(*	=====	LUC	[1]	==========	=	=	*)
		If NOT emC_PPC[PPCNum].LuC[1].In.ComFault	THEN
			emC_PPC[PPCNum].Summary.GCFaultSt	:=	emC_PPC[PPCNum].Summary.GCFaultSt	OR	emC_PPC[PPCNum].LuC[1].In.GCFaultSt	;
			emC_PPC[PPCNum].Summary.NonCriticalAlarm	:=	emC_PPC[PPCNum].Summary.NonCriticalAlarm	OR	emC_PPC[PPCNum].LuC[1].In.NonCriticalAlarm	;
			emC_PPC[PPCNum].Summary.CriticalAlarm	:=	emC_PPC[PPCNum].Summary.CriticalAlarm	OR	emC_PPC[PPCNum].LuC[1].In.CriticalAlarm	;
			emC_PPC[PPCNum].Summary.Warning	:=	emC_PPC[PPCNum].Summary.Warning	OR	emC_PPC[PPCNum].LuC[1].In.Warning	;
			emC_PPC[PPCNum].Summary.StoppingSt	:=	emC_PPC[PPCNum].Summary.StoppingSt	OR	emC_PPC[PPCNum].LuC[1].In.StoppingSt	;
			emC_PPC[PPCNum].Summary.BlackSys	:=	emC_PPC[PPCNum].Summary.BlackSys	OR	emC_PPC[PPCNum].LuC[1].In.BlackSys	;
		END_IF;
		If NOT emC_PPC[PPCNum].LuC[1].In.ComFault	THEN
			emC_PPC[PPCNum].Summary.ComFaultCnt	:=	emC_PPC[PPCNum].Summary.ComFaultCnt	+	1	;
		END_IF;
		If NOT emC_PPC[PPCNum].LuC[1].In.ComFault AND	emC_PPC[PPCNum].LuC[1].In.OnlineSt 	THEN
		
				emC_PPC[PPCNum].Summary.OnlineCnt	:=	emC_PPC[PPCNum].Summary.OnlineCnt	+	1	;
								
				emC_PPC[PPCNum].Summary.AvgTempAct	:=	(emC_PPC[PPCNum].Summary.AvgTempAct	+	emC_PPC[PPCNum].LuC[1].In.TempAct)/INT_TO_REAL(emC_PPC[PPCNum].Summary.OnlineCnt)	;
				emC_PPC[PPCNum].Summary.TotBatPNomMaxAct	:=	emC_PPC[PPCNum].Summary.TotBatPNomMaxAct	+	emC_PPC[PPCNum].LuC[1].In.BatPNomMaxAct	;
				emC_PPC[PPCNum].Summary.TotBatPNomMinAct	:=	emC_PPC[PPCNum].Summary.TotBatPNomMinAct	+	emC_PPC[PPCNum].LuC[1].In.BatPNomMinAct	;
				emC_PPC[PPCNum].Summary.AvgSocPct	:=	(emC_PPC[PPCNum].Summary.AvgSocPct	+	emC_PPC[PPCNum].LuC[1].In.SocPctAct)/INT_TO_REAL(emC_PPC[PPCNum].Summary.OnlineCnt)	;
				emC_PPC[PPCNum].Summary.AvgUAct	:=	(emC_PPC[PPCNum].Summary.AvgUAct	+	emC_PPC[PPCNum].LuC[1].In.UAct)/INT_TO_REAL(emC_PPC[PPCNum].Summary.OnlineCnt)	;
				emC_PPC[PPCNum].Summary.AvgFAct	:=	(emC_PPC[PPCNum].Summary.AvgFAct	+	emC_PPC[PPCNum].LuC[1].In.FAct)/INT_TO_REAL(emC_PPC[PPCNum].Summary.OnlineCnt)	;
				emC_PPC[PPCNum].Summary.TotPAct	:=	emC_PPC[PPCNum].Summary.TotPAct	+	emC_PPC[PPCNum].LuC[1].In.PAct	;
				emC_PPC[PPCNum].Summary.TotQAct	:=	emC_PPC[PPCNum].Summary.TotQAct	+	emC_PPC[PPCNum].LuC[1].In.QAct	;
		
		END_IF	;	
								
								
(*	=====	LUC	[2]	==========	=	=	*)
		If NOT emC_PPC[PPCNum].LuC[2].In.ComFault	THEN						
			emC_PPC[PPCNum].Summary.GCFaultSt	:=	emC_PPC[PPCNum].Summary.GCFaultSt	OR	emC_PPC[PPCNum].LuC[2].In.GCFaultSt	;	
			emC_PPC[PPCNum].Summary.NonCriticalAlarm	:=	emC_PPC[PPCNum].Summary.NonCriticalAlarm	OR	emC_PPC[PPCNum].LuC[2].In.NonCriticalAlarm	;	
			emC_PPC[PPCNum].Summary.CriticalAlarm	:=	emC_PPC[PPCNum].Summary.CriticalAlarm	OR	emC_PPC[PPCNum].LuC[2].In.CriticalAlarm	;	
			emC_PPC[PPCNum].Summary.Warning	:=	emC_PPC[PPCNum].Summary.Warning	OR	emC_PPC[PPCNum].LuC[2].In.Warning	;	
			emC_PPC[PPCNum].Summary.StoppingSt	:=	emC_PPC[PPCNum].Summary.StoppingSt	OR	emC_PPC[PPCNum].LuC[2].In.StoppingSt	;	
			emC_PPC[PPCNum].Summary.BlackSys	:=	emC_PPC[PPCNum].Summary.BlackSys	OR	emC_PPC[PPCNum].LuC[2].In.BlackSys	;	
		END_IF;							
		If NOT emC_PPC[PPCNum].LuC[2].In.ComFault	THEN						
			emC_PPC[PPCNum].Summary.ComFaultCnt	:=	emC_PPC[PPCNum].Summary.ComFaultCnt	+	1	;	
		END_IF;							
		If NOT emC_PPC[PPCNum].LuC[2].In.ComFault AND	emC_PPC[PPCNum].LuC[2].In.OnlineSt 	THEN					
							
				emC_PPC[PPCNum].Summary.OnlineCnt	:=	emC_PPC[PPCNum].Summary.OnlineCnt	+	1	;
							
				emC_PPC[PPCNum].Summary.AvgTempAct	:=	(emC_PPC[PPCNum].Summary.AvgTempAct	+	emC_PPC[PPCNum].LuC[2].In.TempAct)/INT_TO_REAL(emC_PPC[PPCNum].Summary.OnlineCnt)	;
				emC_PPC[PPCNum].Summary.TotBatPNomMaxAct	:=	emC_PPC[PPCNum].Summary.TotBatPNomMaxAct	+	emC_PPC[PPCNum].LuC[2].In.BatPNomMaxAct	;
				emC_PPC[PPCNum].Summary.TotBatPNomMinAct	:=	emC_PPC[PPCNum].Summary.TotBatPNomMinAct	+	emC_PPC[PPCNum].LuC[2].In.BatPNomMinAct	;
				emC_PPC[PPCNum].Summary.AvgSocPct	:=	(emC_PPC[PPCNum].Summary.AvgSocPct	+	emC_PPC[PPCNum].LuC[2].In.SocPctAct)/INT_TO_REAL(emC_PPC[PPCNum].Summary.OnlineCnt)	;
				emC_PPC[PPCNum].Summary.AvgUAct	:=	(emC_PPC[PPCNum].Summary.AvgUAct	+	emC_PPC[PPCNum].LuC[2].In.UAct)/INT_TO_REAL(emC_PPC[PPCNum].Summary.OnlineCnt)	;
				emC_PPC[PPCNum].Summary.AvgFAct	:=	(emC_PPC[PPCNum].Summary.AvgFAct	+	emC_PPC[PPCNum].LuC[2].In.FAct)/INT_TO_REAL(emC_PPC[PPCNum].Summary.OnlineCnt)	;
				emC_PPC[PPCNum].Summary.TotPAct	:=	emC_PPC[PPCNum].Summary.TotPAct	+	emC_PPC[PPCNum].LuC[2].In.PAct	;
				emC_PPC[PPCNum].Summary.TotQAct	:=	emC_PPC[PPCNum].Summary.TotQAct	+	emC_PPC[PPCNum].LuC[2].In.QAct	;
							
		END_IF	;	
								
					
(*	=====	LUC	[3]	==========	=	=	*)
		If NOT emC_PPC[PPCNum].LuC[3].In.ComFault	THEN						
			emC_PPC[PPCNum].Summary.GCFaultSt	:=	emC_PPC[PPCNum].Summary.GCFaultSt	OR	emC_PPC[PPCNum].LuC[3].In.GCFaultSt	;	
			emC_PPC[PPCNum].Summary.NonCriticalAlarm	:=	emC_PPC[PPCNum].Summary.NonCriticalAlarm	OR	emC_PPC[PPCNum].LuC[3].In.NonCriticalAlarm	;	
			emC_PPC[PPCNum].Summary.CriticalAlarm	:=	emC_PPC[PPCNum].Summary.CriticalAlarm	OR	emC_PPC[PPCNum].LuC[3].In.CriticalAlarm	;	
			emC_PPC[PPCNum].Summary.Warning	:=	emC_PPC[PPCNum].Summary.Warning	OR	emC_PPC[PPCNum].LuC[3].In.Warning	;	
			emC_PPC[PPCNum].Summary.StoppingSt	:=	emC_PPC[PPCNum].Summary.StoppingSt	OR	emC_PPC[PPCNum].LuC[3].In.StoppingSt	;	
			emC_PPC[PPCNum].Summary.BlackSys	:=	emC_PPC[PPCNum].Summary.BlackSys	OR	emC_PPC[PPCNum].LuC[3].In.BlackSys	;	
		END_IF;							
		If NOT emC_PPC[PPCNum].LuC[3].In.ComFault	THEN						
			emC_PPC[PPCNum].Summary.ComFaultCnt	:=	emC_PPC[PPCNum].Summary.ComFaultCnt	+	1	;	
		END_IF;							
		If NOT emC_PPC[PPCNum].LuC[3].In.ComFault AND	emC_PPC[PPCNum].LuC[3].In.OnlineSt 	THEN					
							
				emC_PPC[PPCNum].Summary.OnlineCnt	:=	emC_PPC[PPCNum].Summary.OnlineCnt	+	1	;
							
				emC_PPC[PPCNum].Summary.AvgTempAct	:=	(emC_PPC[PPCNum].Summary.AvgTempAct	+	emC_PPC[PPCNum].LuC[3].In.TempAct)/INT_TO_REAL(emC_PPC[PPCNum].Summary.OnlineCnt)	;
				emC_PPC[PPCNum].Summary.TotBatPNomMaxAct	:=	emC_PPC[PPCNum].Summary.TotBatPNomMaxAct	+	emC_PPC[PPCNum].LuC[3].In.BatPNomMaxAct	;
				emC_PPC[PPCNum].Summary.TotBatPNomMinAct	:=	emC_PPC[PPCNum].Summary.TotBatPNomMinAct	+	emC_PPC[PPCNum].LuC[3].In.BatPNomMinAct	;
				emC_PPC[PPCNum].Summary.AvgSocPct	:=	(emC_PPC[PPCNum].Summary.AvgSocPct	+	emC_PPC[PPCNum].LuC[3].In.SocPctAct)/INT_TO_REAL(emC_PPC[PPCNum].Summary.OnlineCnt)	;
				emC_PPC[PPCNum].Summary.AvgUAct	:=	(emC_PPC[PPCNum].Summary.AvgUAct	+	emC_PPC[PPCNum].LuC[3].In.UAct)/INT_TO_REAL(emC_PPC[PPCNum].Summary.OnlineCnt)	;
				emC_PPC[PPCNum].Summary.AvgFAct	:=	(emC_PPC[PPCNum].Summary.AvgFAct	+	emC_PPC[PPCNum].LuC[3].In.FAct)/INT_TO_REAL(emC_PPC[PPCNum].Summary.OnlineCnt)	;
				emC_PPC[PPCNum].Summary.TotPAct	:=	emC_PPC[PPCNum].Summary.TotPAct	+	emC_PPC[PPCNum].LuC[3].In.PAct	;
				emC_PPC[PPCNum].Summary.TotQAct	:=	emC_PPC[PPCNum].Summary.TotQAct	+	emC_PPC[PPCNum].LuC[3].In.QAct	;
							
		END_IF	;		
								
				
(*	=====	LUC	[4]	==========	=	=	*)
		If NOT emC_PPC[PPCNum].LuC[4].In.ComFault	THEN						
			emC_PPC[PPCNum].Summary.GCFaultSt	:=	emC_PPC[PPCNum].Summary.GCFaultSt	OR	emC_PPC[PPCNum].LuC[4].In.GCFaultSt	;	
			emC_PPC[PPCNum].Summary.NonCriticalAlarm	:=	emC_PPC[PPCNum].Summary.NonCriticalAlarm	OR	emC_PPC[PPCNum].LuC[4].In.NonCriticalAlarm	;	
			emC_PPC[PPCNum].Summary.CriticalAlarm	:=	emC_PPC[PPCNum].Summary.CriticalAlarm	OR	emC_PPC[PPCNum].LuC[4].In.CriticalAlarm	;	
			emC_PPC[PPCNum].Summary.Warning	:=	emC_PPC[PPCNum].Summary.Warning	OR	emC_PPC[PPCNum].LuC[4].In.Warning	;	
			emC_PPC[PPCNum].Summary.StoppingSt	:=	emC_PPC[PPCNum].Summary.StoppingSt	OR	emC_PPC[PPCNum].LuC[4].In.StoppingSt	;	
			emC_PPC[PPCNum].Summary.BlackSys	:=	emC_PPC[PPCNum].Summary.BlackSys	OR	emC_PPC[PPCNum].LuC[4].In.BlackSys	;	
		END_IF;							
		If NOT emC_PPC[PPCNum].LuC[4].In.ComFault	THEN						
			emC_PPC[PPCNum].Summary.ComFaultCnt	:=	emC_PPC[PPCNum].Summary.ComFaultCnt	+	1	;	
		END_IF;							
		If NOT emC_PPC[PPCNum].LuC[4].In.ComFault AND	emC_PPC[PPCNum].LuC[4].In.OnlineSt 	THEN					
							
				emC_PPC[PPCNum].Summary.OnlineCnt	:=	emC_PPC[PPCNum].Summary.OnlineCnt	+	1	;
							
				emC_PPC[PPCNum].Summary.AvgTempAct	:=	(emC_PPC[PPCNum].Summary.AvgTempAct	+	emC_PPC[PPCNum].LuC[4].In.TempAct)/INT_TO_REAL(emC_PPC[PPCNum].Summary.OnlineCnt)	;
				emC_PPC[PPCNum].Summary.TotBatPNomMaxAct	:=	emC_PPC[PPCNum].Summary.TotBatPNomMaxAct	+	emC_PPC[PPCNum].LuC[4].In.BatPNomMaxAct	;
				emC_PPC[PPCNum].Summary.TotBatPNomMinAct	:=	emC_PPC[PPCNum].Summary.TotBatPNomMinAct	+	emC_PPC[PPCNum].LuC[4].In.BatPNomMinAct	;
				emC_PPC[PPCNum].Summary.AvgSocPct	:=	(emC_PPC[PPCNum].Summary.AvgSocPct	+	emC_PPC[PPCNum].LuC[4].In.SocPctAct)/INT_TO_REAL(emC_PPC[PPCNum].Summary.OnlineCnt)	;
				emC_PPC[PPCNum].Summary.AvgUAct	:=	(emC_PPC[PPCNum].Summary.AvgUAct	+	emC_PPC[PPCNum].LuC[4].In.UAct)/INT_TO_REAL(emC_PPC[PPCNum].Summary.OnlineCnt)	;
				emC_PPC[PPCNum].Summary.AvgFAct	:=	(emC_PPC[PPCNum].Summary.AvgFAct	+	emC_PPC[PPCNum].LuC[4].In.FAct)/INT_TO_REAL(emC_PPC[PPCNum].Summary.OnlineCnt)	;
				emC_PPC[PPCNum].Summary.TotPAct	:=	emC_PPC[PPCNum].Summary.TotPAct	+	emC_PPC[PPCNum].LuC[4].In.PAct	;
				emC_PPC[PPCNum].Summary.TotQAct	:=	emC_PPC[PPCNum].Summary.TotQAct	+	emC_PPC[PPCNum].LuC[4].In.QAct	;
							
		END_IF	;	
								
					
(*	=====	LUC	[5]	==========	=	=	*)
		If NOT emC_PPC[PPCNum].LuC[5].In.ComFault	THEN						
			emC_PPC[PPCNum].Summary.GCFaultSt	:=	emC_PPC[PPCNum].Summary.GCFaultSt	OR	emC_PPC[PPCNum].LuC[5].In.GCFaultSt	;	
			emC_PPC[PPCNum].Summary.NonCriticalAlarm	:=	emC_PPC[PPCNum].Summary.NonCriticalAlarm	OR	emC_PPC[PPCNum].LuC[5].In.NonCriticalAlarm	;	
			emC_PPC[PPCNum].Summary.CriticalAlarm	:=	emC_PPC[PPCNum].Summary.CriticalAlarm	OR	emC_PPC[PPCNum].LuC[5].In.CriticalAlarm	;	
			emC_PPC[PPCNum].Summary.Warning	:=	emC_PPC[PPCNum].Summary.Warning	OR	emC_PPC[PPCNum].LuC[5].In.Warning	;	
			emC_PPC[PPCNum].Summary.StoppingSt	:=	emC_PPC[PPCNum].Summary.StoppingSt	OR	emC_PPC[PPCNum].LuC[5].In.StoppingSt	;	
			emC_PPC[PPCNum].Summary.BlackSys	:=	emC_PPC[PPCNum].Summary.BlackSys	OR	emC_PPC[PPCNum].LuC[5].In.BlackSys	;	
		END_IF;							
		If NOT emC_PPC[PPCNum].LuC[5].In.ComFault	THEN						
			emC_PPC[PPCNum].Summary.ComFaultCnt	:=	emC_PPC[PPCNum].Summary.ComFaultCnt	+	1	;	
		END_IF;							
		If NOT emC_PPC[PPCNum].LuC[5].In.ComFault AND	emC_PPC[PPCNum].LuC[5].In.OnlineSt 	THEN					
							
				emC_PPC[PPCNum].Summary.OnlineCnt	:=	emC_PPC[PPCNum].Summary.OnlineCnt	+	1	;
							
				emC_PPC[PPCNum].Summary.AvgTempAct	:=	(emC_PPC[PPCNum].Summary.AvgTempAct	+	emC_PPC[PPCNum].LuC[5].In.TempAct)/INT_TO_REAL(emC_PPC[PPCNum].Summary.OnlineCnt)	;
				emC_PPC[PPCNum].Summary.TotBatPNomMaxAct	:=	emC_PPC[PPCNum].Summary.TotBatPNomMaxAct	+	emC_PPC[PPCNum].LuC[5].In.BatPNomMaxAct	;
				emC_PPC[PPCNum].Summary.TotBatPNomMinAct	:=	emC_PPC[PPCNum].Summary.TotBatPNomMinAct	+	emC_PPC[PPCNum].LuC[5].In.BatPNomMinAct	;
				emC_PPC[PPCNum].Summary.AvgSocPct	:=	(emC_PPC[PPCNum].Summary.AvgSocPct	+	emC_PPC[PPCNum].LuC[5].In.SocPctAct)/INT_TO_REAL(emC_PPC[PPCNum].Summary.OnlineCnt)	;
				emC_PPC[PPCNum].Summary.AvgUAct	:=	(emC_PPC[PPCNum].Summary.AvgUAct	+	emC_PPC[PPCNum].LuC[5].In.UAct)/INT_TO_REAL(emC_PPC[PPCNum].Summary.OnlineCnt)	;
				emC_PPC[PPCNum].Summary.AvgFAct	:=	(emC_PPC[PPCNum].Summary.AvgFAct	+	emC_PPC[PPCNum].LuC[5].In.FAct)/INT_TO_REAL(emC_PPC[PPCNum].Summary.OnlineCnt)	;
				emC_PPC[PPCNum].Summary.TotPAct	:=	emC_PPC[PPCNum].Summary.TotPAct	+	emC_PPC[PPCNum].LuC[5].In.PAct	;
				emC_PPC[PPCNum].Summary.TotQAct	:=	emC_PPC[PPCNum].Summary.TotQAct	+	emC_PPC[PPCNum].LuC[5].In.QAct	;
							
		END_IF	;	
								
					
(*	=====	LUC	[6]	==========	=	=	*)
		If NOT emC_PPC[PPCNum].LuC[6].In.ComFault	THEN						
			emC_PPC[PPCNum].Summary.GCFaultSt	:=	emC_PPC[PPCNum].Summary.GCFaultSt	OR	emC_PPC[PPCNum].LuC[6].In.GCFaultSt	;	
			emC_PPC[PPCNum].Summary.NonCriticalAlarm	:=	emC_PPC[PPCNum].Summary.NonCriticalAlarm	OR	emC_PPC[PPCNum].LuC[6].In.NonCriticalAlarm	;	
			emC_PPC[PPCNum].Summary.CriticalAlarm	:=	emC_PPC[PPCNum].Summary.CriticalAlarm	OR	emC_PPC[PPCNum].LuC[6].In.CriticalAlarm	;	
			emC_PPC[PPCNum].Summary.Warning	:=	emC_PPC[PPCNum].Summary.Warning	OR	emC_PPC[PPCNum].LuC[6].In.Warning	;	
			emC_PPC[PPCNum].Summary.StoppingSt	:=	emC_PPC[PPCNum].Summary.StoppingSt	OR	emC_PPC[PPCNum].LuC[6].In.StoppingSt	;	
			emC_PPC[PPCNum].Summary.BlackSys	:=	emC_PPC[PPCNum].Summary.BlackSys	OR	emC_PPC[PPCNum].LuC[6].In.BlackSys	;	
		END_IF;							
		If NOT emC_PPC[PPCNum].LuC[6].In.ComFault	THEN						
			emC_PPC[PPCNum].Summary.ComFaultCnt	:=	emC_PPC[PPCNum].Summary.ComFaultCnt	+	1	;	
		END_IF;							
		If NOT emC_PPC[PPCNum].LuC[6].In.ComFault AND	emC_PPC[PPCNum].LuC[6].In.OnlineSt 	THEN					
							
				emC_PPC[PPCNum].Summary.OnlineCnt	:=	emC_PPC[PPCNum].Summary.OnlineCnt	+	1	;
							
				emC_PPC[PPCNum].Summary.AvgTempAct	:=	(emC_PPC[PPCNum].Summary.AvgTempAct	+	emC_PPC[PPCNum].LuC[6].In.TempAct)/INT_TO_REAL(emC_PPC[PPCNum].Summary.OnlineCnt)	;
				emC_PPC[PPCNum].Summary.TotBatPNomMaxAct	:=	emC_PPC[PPCNum].Summary.TotBatPNomMaxAct	+	emC_PPC[PPCNum].LuC[6].In.BatPNomMaxAct	;
				emC_PPC[PPCNum].Summary.TotBatPNomMinAct	:=	emC_PPC[PPCNum].Summary.TotBatPNomMinAct	+	emC_PPC[PPCNum].LuC[6].In.BatPNomMinAct	;
				emC_PPC[PPCNum].Summary.AvgSocPct	:=	(emC_PPC[PPCNum].Summary.AvgSocPct	+	emC_PPC[PPCNum].LuC[6].In.SocPctAct)/INT_TO_REAL(emC_PPC[PPCNum].Summary.OnlineCnt)	;
				emC_PPC[PPCNum].Summary.AvgUAct	:=	(emC_PPC[PPCNum].Summary.AvgUAct	+	emC_PPC[PPCNum].LuC[6].In.UAct)/INT_TO_REAL(emC_PPC[PPCNum].Summary.OnlineCnt)	;
				emC_PPC[PPCNum].Summary.AvgFAct	:=	(emC_PPC[PPCNum].Summary.AvgFAct	+	emC_PPC[PPCNum].LuC[6].In.FAct)/INT_TO_REAL(emC_PPC[PPCNum].Summary.OnlineCnt)	;
				emC_PPC[PPCNum].Summary.TotPAct	:=	emC_PPC[PPCNum].Summary.TotPAct	+	emC_PPC[PPCNum].LuC[6].In.PAct	;
				emC_PPC[PPCNum].Summary.TotQAct	:=	emC_PPC[PPCNum].Summary.TotQAct	+	emC_PPC[PPCNum].LuC[6].In.QAct	;
							
		END_IF	;	
								
					
(*	=====	LUC	[7]	==========	=	=	*)
		If NOT emC_PPC[PPCNum].LuC[7].In.ComFault	THEN						
			emC_PPC[PPCNum].Summary.GCFaultSt	:=	emC_PPC[PPCNum].Summary.GCFaultSt	OR	emC_PPC[PPCNum].LuC[7].In.GCFaultSt	;	
			emC_PPC[PPCNum].Summary.NonCriticalAlarm	:=	emC_PPC[PPCNum].Summary.NonCriticalAlarm	OR	emC_PPC[PPCNum].LuC[7].In.NonCriticalAlarm	;	
			emC_PPC[PPCNum].Summary.CriticalAlarm	:=	emC_PPC[PPCNum].Summary.CriticalAlarm	OR	emC_PPC[PPCNum].LuC[7].In.CriticalAlarm	;	
			emC_PPC[PPCNum].Summary.Warning	:=	emC_PPC[PPCNum].Summary.Warning	OR	emC_PPC[PPCNum].LuC[7].In.Warning	;	
			emC_PPC[PPCNum].Summary.StoppingSt	:=	emC_PPC[PPCNum].Summary.StoppingSt	OR	emC_PPC[PPCNum].LuC[7].In.StoppingSt	;	
			emC_PPC[PPCNum].Summary.BlackSys	:=	emC_PPC[PPCNum].Summary.BlackSys	OR	emC_PPC[PPCNum].LuC[7].In.BlackSys	;	
		END_IF;							
		If NOT emC_PPC[PPCNum].LuC[7].In.ComFault	THEN						
			emC_PPC[PPCNum].Summary.ComFaultCnt	:=	emC_PPC[PPCNum].Summary.ComFaultCnt	+	1	;	
		END_IF;							
		If NOT emC_PPC[PPCNum].LuC[7].In.ComFault AND	emC_PPC[PPCNum].LuC[7].In.OnlineSt 	THEN					
							
				emC_PPC[PPCNum].Summary.OnlineCnt	:=	emC_PPC[PPCNum].Summary.OnlineCnt	+	1	;
							
				emC_PPC[PPCNum].Summary.AvgTempAct	:=	(emC_PPC[PPCNum].Summary.AvgTempAct	+	emC_PPC[PPCNum].LuC[7].In.TempAct)/INT_TO_REAL(emC_PPC[PPCNum].Summary.OnlineCnt)	;
				emC_PPC[PPCNum].Summary.TotBatPNomMaxAct	:=	emC_PPC[PPCNum].Summary.TotBatPNomMaxAct	+	emC_PPC[PPCNum].LuC[7].In.BatPNomMaxAct	;
				emC_PPC[PPCNum].Summary.TotBatPNomMinAct	:=	emC_PPC[PPCNum].Summary.TotBatPNomMinAct	+	emC_PPC[PPCNum].LuC[7].In.BatPNomMinAct	;
				emC_PPC[PPCNum].Summary.AvgSocPct	:=	(emC_PPC[PPCNum].Summary.AvgSocPct	+	emC_PPC[PPCNum].LuC[7].In.SocPctAct)/INT_TO_REAL(emC_PPC[PPCNum].Summary.OnlineCnt)	;
				emC_PPC[PPCNum].Summary.AvgUAct	:=	(emC_PPC[PPCNum].Summary.AvgUAct	+	emC_PPC[PPCNum].LuC[7].In.UAct)/INT_TO_REAL(emC_PPC[PPCNum].Summary.OnlineCnt)	;
				emC_PPC[PPCNum].Summary.AvgFAct	:=	(emC_PPC[PPCNum].Summary.AvgFAct	+	emC_PPC[PPCNum].LuC[7].In.FAct)/INT_TO_REAL(emC_PPC[PPCNum].Summary.OnlineCnt)	;
				emC_PPC[PPCNum].Summary.TotPAct	:=	emC_PPC[PPCNum].Summary.TotPAct	+	emC_PPC[PPCNum].LuC[7].In.PAct	;
				emC_PPC[PPCNum].Summary.TotQAct	:=	emC_PPC[PPCNum].Summary.TotQAct	+	emC_PPC[PPCNum].LuC[7].In.QAct	;
							
		END_IF	;
								
						
(*	=====	LUC	[8]	==========	=	=	*)
		If NOT emC_PPC[PPCNum].LuC[8].In.ComFault	THEN						
			emC_PPC[PPCNum].Summary.GCFaultSt	:=	emC_PPC[PPCNum].Summary.GCFaultSt	OR	emC_PPC[PPCNum].LuC[8].In.GCFaultSt	;	
			emC_PPC[PPCNum].Summary.NonCriticalAlarm	:=	emC_PPC[PPCNum].Summary.NonCriticalAlarm	OR	emC_PPC[PPCNum].LuC[8].In.NonCriticalAlarm	;	
			emC_PPC[PPCNum].Summary.CriticalAlarm	:=	emC_PPC[PPCNum].Summary.CriticalAlarm	OR	emC_PPC[PPCNum].LuC[8].In.CriticalAlarm	;	
			emC_PPC[PPCNum].Summary.Warning	:=	emC_PPC[PPCNum].Summary.Warning	OR	emC_PPC[PPCNum].LuC[8].In.Warning	;	
			emC_PPC[PPCNum].Summary.StoppingSt	:=	emC_PPC[PPCNum].Summary.StoppingSt	OR	emC_PPC[PPCNum].LuC[8].In.StoppingSt	;	
			emC_PPC[PPCNum].Summary.BlackSys	:=	emC_PPC[PPCNum].Summary.BlackSys	OR	emC_PPC[PPCNum].LuC[8].In.BlackSys	;	
		END_IF;							
		If NOT emC_PPC[PPCNum].LuC[8].In.ComFault	THEN						
			emC_PPC[PPCNum].Summary.ComFaultCnt	:=	emC_PPC[PPCNum].Summary.ComFaultCnt	+	1	;	
		END_IF;							
		If NOT emC_PPC[PPCNum].LuC[8].In.ComFault AND	emC_PPC[PPCNum].LuC[8].In.OnlineSt 	THEN					
							
				emC_PPC[PPCNum].Summary.OnlineCnt	:=	emC_PPC[PPCNum].Summary.OnlineCnt	+	1	;
							
				emC_PPC[PPCNum].Summary.AvgTempAct	:=	(emC_PPC[PPCNum].Summary.AvgTempAct	+	emC_PPC[PPCNum].LuC[8].In.TempAct)/INT_TO_REAL(emC_PPC[PPCNum].Summary.OnlineCnt)	;
				emC_PPC[PPCNum].Summary.TotBatPNomMaxAct	:=	emC_PPC[PPCNum].Summary.TotBatPNomMaxAct	+	emC_PPC[PPCNum].LuC[8].In.BatPNomMaxAct	;
				emC_PPC[PPCNum].Summary.TotBatPNomMinAct	:=	emC_PPC[PPCNum].Summary.TotBatPNomMinAct	+	emC_PPC[PPCNum].LuC[8].In.BatPNomMinAct	;
				emC_PPC[PPCNum].Summary.AvgSocPct	:=	(emC_PPC[PPCNum].Summary.AvgSocPct	+	emC_PPC[PPCNum].LuC[8].In.SocPctAct)/INT_TO_REAL(emC_PPC[PPCNum].Summary.OnlineCnt)	;
				emC_PPC[PPCNum].Summary.AvgUAct	:=	(emC_PPC[PPCNum].Summary.AvgUAct	+	emC_PPC[PPCNum].LuC[8].In.UAct)/INT_TO_REAL(emC_PPC[PPCNum].Summary.OnlineCnt)	;
				emC_PPC[PPCNum].Summary.AvgFAct	:=	(emC_PPC[PPCNum].Summary.AvgFAct	+	emC_PPC[PPCNum].LuC[8].In.FAct)/INT_TO_REAL(emC_PPC[PPCNum].Summary.OnlineCnt)	;
				emC_PPC[PPCNum].Summary.TotPAct	:=	emC_PPC[PPCNum].Summary.TotPAct	+	emC_PPC[PPCNum].LuC[8].In.PAct	;
				emC_PPC[PPCNum].Summary.TotQAct	:=	emC_PPC[PPCNum].Summary.TotQAct	+	emC_PPC[PPCNum].LuC[8].In.QAct	;
							
		END_IF	;
							
						
					
END_PROGRAM

PROGRAM emC_PPC_R05_MSH_Out
  VAR
    RTU_RTC_1 : RTU_RTC;
  END_VAR
  VAR_EXTERNAL
    Execute_Cmd : BOOL;
    LuCNum : INT;
  END_VAR
  VAR
    Timestamp : Timestamp;
  END_VAR
  VAR_EXTERNAL
    emC_LUC : emC_LUC_Array;
    PPCNum : INT;
    emC_PPC : emC_PPC_Array;
  END_VAR
  VAR
    i : INT;
    NetOnlineSt : BOOL;
    NetIslandReq : BOOL;
    AutoStartCmd : BOOL;
    AutoStopCmd : BOOL;
    TON_1 : TON;
    NextStart : INT;
    FSetOut : REAL := 50.0;
    USetOut : REAL := 480.0;
    PSetOut : REAL;
    QSetOut : REAL;
    FAct : REAL;
    UAct : REAL;
    PAct : REAL;
    QAct : REAL;
    FAct_temp : REAL;
    UAct_temp : REAL;
    AutoStopCmd_1 : BOOL;
    AutoStopCmd_2 : BOOL;
    AutoStopCmd_3 : BOOL;
    AutoStopCmd_4 : BOOL;
    AutoStopCmd_5 : BOOL;
    emC_PPC_LuCOut_1 : emC_PPC_LuCOut;
    L1_FSetOut_I : FSO;
    L1_USetOut_I : FSO;
    L1_PSetOut_I : FSO;
    L1_QSetOut_I : FSO;
    L1_FastFSetOut_I : FSO;
    L1_FastUSetOut_I : FSO;
    L1_FastPSetOut_I : FSO;
    L1_FastQSetOut_I : FSO;
    L1_FastF_SF_I : FSO;
    L1_FastU_SF_I : FSO;
    L1_FastP_SF_I : FSO;
    L1_FastQ_SF_I : FSO;
    L1_FSetOut_Q : FSO;
    L1_USetOut_Q : FSO;
    L1_PSetOut_Q : FSO;
    L1_QSetOut_Q : FSO;
    L1_FastFSetOut_Q : FSO;
    L1_FastUSetOut_Q : FSO;
    L1_FastPSetOut_Q : FSO;
    L1_FastQSetOut_Q : FSO;
    L1_FastF_SF_Q : FSO;
    L1_FastU_SF_Q : FSO;
    L1_FastP_SF_Q : FSO;
    L1_FastQ_SF_Q : FSO;
    L1_NetOnlineSt_I : SCO;
    L1_NetIslandReq_I : SCO;
    L1_AutoStartCmd_I : SCO;
    L1_AutoStopCmd_I : SCO;
    L1_StopRampSt_I : SCO;
    L1_NetOnlineSt_Q : SCO;
    L1_NetIslandReq_Q : SCO;
    L1_AutoStartCmd_Q : SCO;
    L1_AutoStopCmd_Q : SCO;
    L1_StopRampSt_Q : SCO;
    emC_PPC_LuCOut_2 : emC_PPC_LuCOut;
    L4_FSetOut_I : FSO;
    L4_USetOut_I : FSO;
    L4_PSetOut_I : FSO;
    L4_QSetOut_I : FSO;
    L4_FastFSetOut_I : FSO;
    L4_FastUSetOut_I : FSO;
    L4_FastPSetOut_I : FSO;
    L4_FastQSetOut_I : FSO;
    L4_FastF_SF_I : FSO;
    L4_FastU_SF_I : FSO;
    L4_FastP_SF_I : FSO;
    L4_FastQ_SF_I : FSO;
    L4_FSetOut_Q : FSO;
    L4_USetOut_Q : FSO;
    L4_PSetOut_Q : FSO;
    L4_QSetOut_Q : FSO;
    L4_FastFSetOut_Q : FSO;
    L4_FastUSetOut_Q : FSO;
    L4_FastPSetOut_Q : FSO;
    L4_FastQSetOut_Q : FSO;
    L4_FastF_SF_Q : FSO;
    L4_FastU_SF_Q : FSO;
    L4_FastP_SF_Q : FSO;
    L4_FastQ_SF_Q : FSO;
    L4_NetOnlineSt_I : SCO;
    L4_NetIslandReq_I : SCO;
    L4_AutoStartCmd_I : SCO;
    L4_AutoStopCmd_I : SCO;
    L4_StopRampSt_I : SCO;
    L4_NetOnlineSt_Q : SCO;
    L4_NetIslandReq_Q : SCO;
    L4_AutoStartCmd_Q : SCO;
    L4_AutoStopCmd_Q : SCO;
    L4_StopRampSt_Q : SCO;
    L3_FSetOut_I : FSO;
    L3_USetOut_I : FSO;
    L3_PSetOut_I : FSO;
    L3_QSetOut_I : FSO;
    L3_FastFSetOut_I : FSO;
    L3_FastUSetOut_I : FSO;
    L3_FastPSetOut_I : FSO;
    L3_FastQSetOut_I : FSO;
    L3_FastF_SF_I : FSO;
    L3_FastU_SF_I : FSO;
    L3_FastP_SF_I : FSO;
    L3_FastQ_SF_I : FSO;
    L3_NetOnlineSt_I : SCO;
    L3_NetIslandReq_I : SCO;
    L3_AutoStartCmd_I : SCO;
    L3_AutoStopCmd_I : SCO;
    L3_StopRampSt_I : SCO;
    L3_FSetOut_Q : FSO;
    L3_USetOut_Q : FSO;
    L3_PSetOut_Q : FSO;
    L3_QSetOut_Q : FSO;
    L3_NetOnlineSt_Q : SCO;
    L3_NetIslandReq_Q : SCO;
    L3_AutoStartCmd_Q : SCO;
    L3_AutoStopCmd_Q : SCO;
    L3_StopRampSt_Q : SCO;
    L3_FastFSetOut_Q : FSO;
    L3_FastUSetOut_Q : FSO;
    L3_FastPSetOut_Q : FSO;
    L3_FastQSetOut_Q : FSO;
    L3_FastF_SF_Q : FSO;
    L3_FastU_SF_Q : FSO;
    L3_FastP_SF_Q : FSO;
    L3_FastQ_SF_Q : FSO;
    emC_PPC_LuCOut_3 : emC_PPC_LuCOut;
    emC_PPC_LuCOut_4 : emC_PPC_LuCOut;
    L2_FSetOut_I : FSO;
    L2_USetOut_I : FSO;
    L2_PSetOut_I : FSO;
    L2_QSetOut_I : FSO;
    L2_FastFSetOut_I : FSO;
    L2_FastUSetOut_I : FSO;
    L2_FastPSetOut_I : FSO;
    L2_FastQSetOut_I : FSO;
    L2_FastF_SF_I : FSO;
    L2_FastU_SF_I : FSO;
    L2_FastP_SF_I : FSO;
    L2_FastQ_SF_I : FSO;
    L2_FSetOut_Q : FSO;
    L2_USetOut_Q : FSO;
    L2_PSetOut_Q : FSO;
    L2_QSetOut_Q : FSO;
    L2_FastFSetOut_Q : FSO;
    L2_FastUSetOut_Q : FSO;
    L2_FastPSetOut_Q : FSO;
    L2_FastQSetOut_Q : FSO;
    L2_FastF_SF_Q : FSO;
    L2_FastU_SF_Q : FSO;
    L2_FastP_SF_Q : FSO;
    L2_FastQ_SF_Q : FSO;
    L2_NetOnlineSt_I : SCO;
    L2_NetIslandReq_I : SCO;
    L2_AutoStartCmd_I : SCO;
    L2_AutoStopCmd_I : SCO;
    L2_StopRampSt_I : SCO;
    L2_NetOnlineSt_Q : SCO;
    L2_NetIslandReq_Q : SCO;
    L2_AutoStartCmd_Q : SCO;
    L2_AutoStopCmd_Q : SCO;
    L2_StopRampSt_Q : SCO;
    emC_PPC_LuCOut_5 : emC_PPC_LuCOut;
    L5_FSetOut_I : FSO;
    L5_USetOut_I : FSO;
    L5_PSetOut_I : FSO;
    L5_QSetOut_I : FSO;
    L5_FastFSetOut_I : FSO;
    L5_FastUSetOut_I : FSO;
    L5_FastPSetOut_I : FSO;
    L5_FastQSetOut_I : FSO;
    L5_FastF_SF_I : FSO;
    L5_FastU_SF_I : FSO;
    L5_FastP_SF_I : FSO;
    L5_FastQ_SF_I : FSO;
    L5_FSetOut_Q : FSO;
    L5_USetOut_Q : FSO;
    L5_PSetOut_Q : FSO;
    L5_QSetOut_Q : FSO;
    L5_FastFSetOut_Q : FSO;
    L5_FastUSetOut_Q : FSO;
    L5_FastPSetOut_Q : FSO;
    L5_FastQSetOut_Q : FSO;
    L5_FastF_SF_Q : FSO;
    L5_FastU_SF_Q : FSO;
    L5_FastP_SF_Q : FSO;
    L5_FastQ_SF_Q : FSO;
    L5_NetOnlineSt_I : SCO;
    L5_NetIslandReq_I : SCO;
    L5_AutoStartCmd_I : SCO;
    L5_AutoStopCmd_I : SCO;
    L5_StopRampSt_I : SCO;
    L5_NetOnlineSt_Q : SCO;
    L5_NetIslandReq_Q : SCO;
    L5_AutoStartCmd_Q : SCO;
    L5_AutoStopCmd_Q : SCO;
    L5_StopRampSt_Q : SCO;
  END_VAR

						
							RTU_RTC_1(EN:=TRUE);
Timestamp.Milliseconds :=RTU_RTC_1.Milliseconds;
Timestamp.Minutes :=RTU_RTC_1.Minutes;
Timestamp.IV :=RTU_RTC_1.IV;
Timestamp.Hours :=RTU_RTC_1.Hours;
Timestamp.Summertime :=RTU_RTC_1.Summertime;
Timestamp.DayOfMonth :=RTU_RTC_1.DayOfMonth;
Timestamp.DayOfWeek :=RTU_RTC_1.DayOfWeek;
Timestamp.Month :=RTU_RTC_1.Months;
Timestamp.Year :=RTU_RTC_1.Year;
								
Execute_Cmd:= Sel(Execute_Cmd, TRUE,FALSE)	;
							
							
							
								
(*____________________________________________________*)
FAct_temp := 0.0;
UAct_temp := 0.0;
PAct:=  0.0;
QAct :=  0.0;
								
TON_1(IN:=not TON_1.Q,PT:=t#5s);
								
if TON_1.Q and AutoStartCmd and (NextStart < LuCNum) then NextStart := NextStart + 1; AutoStartCmd := FALSE; End_IF;
								
for i:= 1 to LuCNum do
	emC_PPC[PPCNum].LuC[i].Out.NetOnlineSt := NetOnlineSt;
	emC_PPC[PPCNum].LuC[i].Out.NetIslandReq := NetIslandReq;
	emC_PPC[PPCNum].LuC[i].Out.AutoStartCmd := i <= NextStart;
	emC_PPC[PPCNum].LuC[i].Out.FSetOut	:=	FSetOut;
	emC_PPC[PPCNum].LuC[i].Out.USetOut	:=	USetOut;
	emC_PPC[PPCNum].LuC[i].Out.PSetOut	:=	PSetOut;
	emC_PPC[PPCNum].LuC[i].Out.QSetOut	:=QSetOut;
								
	FAct_temp := (emC_PPC[PPCNum].LuC[i].In.FAct + FAct_temp) ;
	UAct_temp := (emC_PPC[PPCNum].LuC[i].In.UAct + UAct_temp);
	PAct:= emC_PPC[PPCNum].LuC[i].In.PAct + PAct;
	QAct :=emC_PPC[PPCNum].LuC[i].In.QAct + QAct;
End_For;
								
FAct := FAct_temp / int_to_Real(LuCNum);
UAct :=  UAct_temp /  int_to_Real(LuCNum);
								
								
								
emC_PPC[PPCNum].LuC[1].Out.AutoStopCmd := AutoStopCmd_1;
emC_PPC[PPCNum].LuC[2].Out.AutoStopCmd := AutoStopCmd_2;
emC_PPC[PPCNum].LuC[3].Out.AutoStopCmd := AutoStopCmd_3;
emC_PPC[PPCNum].LuC[4].Out.AutoStopCmd := AutoStopCmd_4;
emC_PPC[PPCNum].LuC[5].Out.AutoStopCmd := AutoStopCmd_5;
							
							LuCNum	:=	1	;
emC_PPC_LuCOut_1(									
				FastSlowDataEnPa		:=	emC_PPC[PPCNum].Param.FastSlowDataEnPa	,
				FSetOut		:=	emC_PPC[PPCNum].LuC[LuCNum].Out.FSetOut	,	
				USetOut		:=	emC_PPC[PPCNum].LuC[LuCNum].Out.USetOut	,	
				PSetOut		:=	emC_PPC[PPCNum].LuC[LuCNum].Out.PSetOut	,	
				QSetOut		:=	emC_PPC[PPCNum].LuC[LuCNum].Out.QSetOut	,	
				F_SF		:=	emC_PPC[PPCNum].LuC[LuCNum].Out.F_SF	,	
				U_SF		:=	emC_PPC[PPCNum].LuC[LuCNum].Out.U_SF	,	
				P_SF		:=	emC_PPC[PPCNum].LuC[LuCNum].Out.P_SF	,	
				Q_SF		:=	emC_PPC[PPCNum].LuC[LuCNum].Out.Q_SF	,
				NetOnlineSt	:=	emC_PPC[PPCNum].LuC[LuCNum].Out.NetOnlineSt	,					
				NetIslandReq:=	emC_PPC[PPCNum].LuC[LuCNum].Out.NetIslandReq	,					
				AutoStartCmd:=	emC_PPC[PPCNum].LuC[LuCNum].Out.AutoStartCmd	,					
				AutoStopCmd	:=	emC_PPC[PPCNum].LuC[LuCNum].Out.AutoStopCmd	,
				
				PQFVSelPaGfw:=emC_PPC[PPCNum].Param.PQFVSelPaGfw	,
				PQFVSelPaGfm:=emC_PPC[PPCNum].Param.PQFVSelPaGfm	,
				AllowGFWEnPa:=emC_PPC[PPCNum].Param.AllowGFWEnPa	,
				AllowGFMEnPa:=emC_PPC[PPCNum].Param.AllowGFMEnPa	,
				BlackSys	:=  emC_PPC[PPCNum].LuC[LuCNum].Out.BlackSys	
				)	;
								
								
									
	L1_FSetOut_Q	:=	emC_PPC_LuCOut_1.FSetOut_Q	;					
	L1_USetOut_Q	:=	emC_PPC_LuCOut_1.USetOut_Q	;					
	L1_PSetOut_Q	:=	emC_PPC_LuCOut_1.PSetOut_Q	;					
	L1_QSetOut_Q	:=	emC_PPC_LuCOut_1.QSetOut_Q	;					
	L1_FastFSetOut_Q	:=	emC_PPC_LuCOut_1.FastFSetOut_Q	;					
	L1_FastUSetOut_Q	:=	emC_PPC_LuCOut_1.FastUSetOut_Q	;					
	L1_FastPSetOut_Q	:=	emC_PPC_LuCOut_1.FastPSetOut_Q	;					
	L1_FastQSetOut_Q	:=	emC_PPC_LuCOut_1.FastQSetOut_Q	;					
	L1_FastF_SF_Q	:=	emC_PPC_LuCOut_1.FastF_SF_Q	;					
	L1_FastU_SF_Q	:=	emC_PPC_LuCOut_1.FastU_SF_Q	;					
	L1_FastP_SF_Q	:=	emC_PPC_LuCOut_1.FastP_SF_Q	;							
	L1_NetOnlineSt_Q	:=	emC_PPC_LuCOut_1.NetOnlineSt_Q	;					
	L1_NetIslandReq_Q	:=	emC_PPC_LuCOut_1.NetIslandReq_Q	;					
	L1_AutoStartCmd_Q	:=	emC_PPC_LuCOut_1.AutoStartCmd_Q	;					
	L1_AutoStopCmd_Q	:=	emC_PPC_LuCOut_1.AutoStopCmd_Q	;
							
							LuCNum	:=	LuCNum	+1	;
emC_PPC_LuCOut_2(									
				FastSlowDataEnPa		:=	emC_PPC[PPCNum].Param.FastSlowDataEnPa	,
				FSetOut		:=	emC_PPC[PPCNum].LuC[LuCNum].Out.FSetOut	,	
				USetOut		:=	emC_PPC[PPCNum].LuC[LuCNum].Out.USetOut	,	
				PSetOut		:=	emC_PPC[PPCNum].LuC[LuCNum].Out.PSetOut	,	
				QSetOut		:=	emC_PPC[PPCNum].LuC[LuCNum].Out.QSetOut	,	
				F_SF		:=	emC_PPC[PPCNum].LuC[LuCNum].Out.F_SF	,	
				U_SF		:=	emC_PPC[PPCNum].LuC[LuCNum].Out.U_SF	,	
				P_SF		:=	emC_PPC[PPCNum].LuC[LuCNum].Out.P_SF	,	
				Q_SF		:=	emC_PPC[PPCNum].LuC[LuCNum].Out.Q_SF	,
				NetOnlineSt	:=	emC_PPC[PPCNum].LuC[LuCNum].Out.NetOnlineSt	,					
				NetIslandReq:=	emC_PPC[PPCNum].LuC[LuCNum].Out.NetIslandReq	,					
				AutoStartCmd:=	emC_PPC[PPCNum].LuC[LuCNum].Out.AutoStartCmd	,					
				AutoStopCmd	:=	emC_PPC[PPCNum].LuC[LuCNum].Out.AutoStopCmd	,
				
				PQFVSelPaGfw:=emC_PPC[PPCNum].Param.PQFVSelPaGfw	,
				PQFVSelPaGfm:=emC_PPC[PPCNum].Param.PQFVSelPaGfm	,
				AllowGFWEnPa:=emC_PPC[PPCNum].Param.AllowGFWEnPa	,
				AllowGFMEnPa:=emC_PPC[PPCNum].Param.AllowGFMEnPa	,
				BlackSys	:=  emC_PPC[PPCNum].LuC[LuCNum].Out.BlackSys	
				)	;
								
								
									
	L2_FSetOut_Q	:=	emC_PPC_LuCOut_2.FSetOut_Q	;					
	L2_USetOut_Q	:=	emC_PPC_LuCOut_2.USetOut_Q	;					
	L2_PSetOut_Q	:=	emC_PPC_LuCOut_2.PSetOut_Q	;					
	L2_QSetOut_Q	:=	emC_PPC_LuCOut_2.QSetOut_Q	;					
	L2_FastFSetOut_Q	:=	emC_PPC_LuCOut_2.FastFSetOut_Q	;					
	L2_FastUSetOut_Q	:=	emC_PPC_LuCOut_2.FastUSetOut_Q	;					
	L2_FastPSetOut_Q	:=	emC_PPC_LuCOut_2.FastPSetOut_Q	;					
	L2_FastQSetOut_Q	:=	emC_PPC_LuCOut_2.FastQSetOut_Q	;					
	L2_FastF_SF_Q	:=	emC_PPC_LuCOut_2.FastF_SF_Q	;					
	L2_FastU_SF_Q	:=	emC_PPC_LuCOut_2.FastU_SF_Q	;					
	L2_FastP_SF_Q	:=	emC_PPC_LuCOut_2.FastP_SF_Q	;							
	L2_NetOnlineSt_Q	:=	emC_PPC_LuCOut_2.NetOnlineSt_Q	;					
	L2_NetIslandReq_Q	:=	emC_PPC_LuCOut_2.NetIslandReq_Q	;					
	L2_AutoStartCmd_Q	:=	emC_PPC_LuCOut_2.AutoStartCmd_Q	;					
	L2_AutoStopCmd_Q	:=	emC_PPC_LuCOut_2.AutoStopCmd_Q	;
							
							LuCNum	:=	LuCNum	+1	;
emC_PPC_LuCOut_3(									
				FastSlowDataEnPa		:=	emC_PPC[PPCNum].Param.FastSlowDataEnPa	,
				FSetOut		:=	emC_PPC[PPCNum].LuC[LuCNum].Out.FSetOut	,	
				USetOut		:=	emC_PPC[PPCNum].LuC[LuCNum].Out.USetOut	,	
				PSetOut		:=	emC_PPC[PPCNum].LuC[LuCNum].Out.PSetOut	,	
				QSetOut		:=	emC_PPC[PPCNum].LuC[LuCNum].Out.QSetOut	,	
				F_SF		:=	emC_PPC[PPCNum].LuC[LuCNum].Out.F_SF	,	
				U_SF		:=	emC_PPC[PPCNum].LuC[LuCNum].Out.U_SF	,	
				P_SF		:=	emC_PPC[PPCNum].LuC[LuCNum].Out.P_SF	,	
				Q_SF		:=	emC_PPC[PPCNum].LuC[LuCNum].Out.Q_SF	,
				NetOnlineSt	:=	emC_PPC[PPCNum].LuC[LuCNum].Out.NetOnlineSt	,					
				NetIslandReq:=	emC_PPC[PPCNum].LuC[LuCNum].Out.NetIslandReq	,					
				AutoStartCmd:=	emC_PPC[PPCNum].LuC[LuCNum].Out.AutoStartCmd	,					
				AutoStopCmd	:=	emC_PPC[PPCNum].LuC[LuCNum].Out.AutoStopCmd	,
				
				PQFVSelPaGfw:=emC_PPC[PPCNum].Param.PQFVSelPaGfw	,
				PQFVSelPaGfm:=emC_PPC[PPCNum].Param.PQFVSelPaGfm	,
				AllowGFWEnPa:=emC_PPC[PPCNum].Param.AllowGFWEnPa	,
				AllowGFMEnPa:=emC_PPC[PPCNum].Param.AllowGFMEnPa	,
				BlackSys	:=  emC_PPC[PPCNum].LuC[LuCNum].Out.BlackSys	
				)	;
								
								
									
	L3_FSetOut_Q	:=	emC_PPC_LuCOut_3.FSetOut_Q	;					
	L3_USetOut_Q	:=	emC_PPC_LuCOut_3.USetOut_Q	;					
	L3_PSetOut_Q	:=	emC_PPC_LuCOut_3.PSetOut_Q	;					
	L3_QSetOut_Q	:=	emC_PPC_LuCOut_3.QSetOut_Q	;					
	L3_FastFSetOut_Q	:=	emC_PPC_LuCOut_3.FastFSetOut_Q	;					
	L3_FastUSetOut_Q	:=	emC_PPC_LuCOut_3.FastUSetOut_Q	;					
	L3_FastPSetOut_Q	:=	emC_PPC_LuCOut_3.FastPSetOut_Q	;					
	L3_FastQSetOut_Q	:=	emC_PPC_LuCOut_3.FastQSetOut_Q	;					
	L3_FastF_SF_Q	:=	emC_PPC_LuCOut_3.FastF_SF_Q	;					
	L3_FastU_SF_Q	:=	emC_PPC_LuCOut_3.FastU_SF_Q	;					
	L3_FastP_SF_Q	:=	emC_PPC_LuCOut_3.FastP_SF_Q	;							
	L3_NetOnlineSt_Q	:=	emC_PPC_LuCOut_3.NetOnlineSt_Q	;					
	L3_NetIslandReq_Q	:=	emC_PPC_LuCOut_3.NetIslandReq_Q	;					
	L3_AutoStartCmd_Q	:=	emC_PPC_LuCOut_3.AutoStartCmd_Q	;					
	L3_AutoStopCmd_Q	:=	emC_PPC_LuCOut_3.AutoStopCmd_Q	;
							
							LuCNum	:=	LuCNum	+1	;
emC_PPC_LuCOut_4(									
				FastSlowDataEnPa		:=	emC_PPC[PPCNum].Param.FastSlowDataEnPa	,
				FSetOut		:=	emC_PPC[PPCNum].LuC[LuCNum].Out.FSetOut	,	
				USetOut		:=	emC_PPC[PPCNum].LuC[LuCNum].Out.USetOut	,	
				PSetOut		:=	emC_PPC[PPCNum].LuC[LuCNum].Out.PSetOut	,	
				QSetOut		:=	emC_PPC[PPCNum].LuC[LuCNum].Out.QSetOut	,	
				F_SF		:=	emC_PPC[PPCNum].LuC[LuCNum].Out.F_SF	,	
				U_SF		:=	emC_PPC[PPCNum].LuC[LuCNum].Out.U_SF	,	
				P_SF		:=	emC_PPC[PPCNum].LuC[LuCNum].Out.P_SF	,	
				Q_SF		:=	emC_PPC[PPCNum].LuC[LuCNum].Out.Q_SF	,
				NetOnlineSt	:=	emC_PPC[PPCNum].LuC[LuCNum].Out.NetOnlineSt	,					
				NetIslandReq:=	emC_PPC[PPCNum].LuC[LuCNum].Out.NetIslandReq	,					
				AutoStartCmd:=	emC_PPC[PPCNum].LuC[LuCNum].Out.AutoStartCmd	,					
				AutoStopCmd	:=	emC_PPC[PPCNum].LuC[LuCNum].Out.AutoStopCmd	,
				
				PQFVSelPaGfw:=emC_PPC[PPCNum].Param.PQFVSelPaGfw	,
				PQFVSelPaGfm:=emC_PPC[PPCNum].Param.PQFVSelPaGfm	,
				AllowGFWEnPa:=emC_PPC[PPCNum].Param.AllowGFWEnPa	,
				AllowGFMEnPa:=emC_PPC[PPCNum].Param.AllowGFMEnPa	,
				BlackSys	:=  emC_PPC[PPCNum].LuC[LuCNum].Out.BlackSys	
				)	;
								
								
									
	L4_FSetOut_Q	:=	emC_PPC_LuCOut_4.FSetOut_Q	;					
	L4_USetOut_Q	:=	emC_PPC_LuCOut_4.USetOut_Q	;					
	L4_PSetOut_Q	:=	emC_PPC_LuCOut_4.PSetOut_Q	;					
	L4_QSetOut_Q	:=	emC_PPC_LuCOut_4.QSetOut_Q	;					
	L4_FastFSetOut_Q	:=	emC_PPC_LuCOut_4.FastFSetOut_Q	;					
	L4_FastUSetOut_Q	:=	emC_PPC_LuCOut_4.FastUSetOut_Q	;					
	L4_FastPSetOut_Q	:=	emC_PPC_LuCOut_4.FastPSetOut_Q	;					
	L4_FastQSetOut_Q	:=	emC_PPC_LuCOut_4.FastQSetOut_Q	;					
	L4_FastF_SF_Q	:=	emC_PPC_LuCOut_4.FastF_SF_Q	;					
	L4_FastU_SF_Q	:=	emC_PPC_LuCOut_4.FastU_SF_Q	;					
	L4_FastP_SF_Q	:=	emC_PPC_LuCOut_4.FastP_SF_Q	;							
	L4_NetOnlineSt_Q	:=	emC_PPC_LuCOut_4.NetOnlineSt_Q	;					
	L4_NetIslandReq_Q	:=	emC_PPC_LuCOut_4.NetIslandReq_Q	;					
	L4_AutoStartCmd_Q	:=	emC_PPC_LuCOut_4.AutoStartCmd_Q	;					
	L4_AutoStopCmd_Q	:=	emC_PPC_LuCOut_4.AutoStopCmd_Q	;
							
							LuCNum	:=	LuCNum	+1	;
emC_PPC_LuCOut_5(									
				FastSlowDataEnPa		:=	emC_PPC[PPCNum].Param.FastSlowDataEnPa	,
				FSetOut		:=	emC_PPC[PPCNum].LuC[LuCNum].Out.FSetOut	,	
				USetOut		:=	emC_PPC[PPCNum].LuC[LuCNum].Out.USetOut	,	
				PSetOut		:=	emC_PPC[PPCNum].LuC[LuCNum].Out.PSetOut	,	
				QSetOut		:=	emC_PPC[PPCNum].LuC[LuCNum].Out.QSetOut	,	
				F_SF		:=	emC_PPC[PPCNum].LuC[LuCNum].Out.F_SF	,	
				U_SF		:=	emC_PPC[PPCNum].LuC[LuCNum].Out.U_SF	,	
				P_SF		:=	emC_PPC[PPCNum].LuC[LuCNum].Out.P_SF	,	
				Q_SF		:=	emC_PPC[PPCNum].LuC[LuCNum].Out.Q_SF	,
				NetOnlineSt	:=	emC_PPC[PPCNum].LuC[LuCNum].Out.NetOnlineSt	,					
				NetIslandReq:=	emC_PPC[PPCNum].LuC[LuCNum].Out.NetIslandReq	,					
				AutoStartCmd:=	emC_PPC[PPCNum].LuC[LuCNum].Out.AutoStartCmd	,					
				AutoStopCmd	:=	emC_PPC[PPCNum].LuC[LuCNum].Out.AutoStopCmd	,
				
				PQFVSelPaGfw:=emC_PPC[PPCNum].Param.PQFVSelPaGfw	,
				PQFVSelPaGfm:=emC_PPC[PPCNum].Param.PQFVSelPaGfm	,
				AllowGFWEnPa:=emC_PPC[PPCNum].Param.AllowGFWEnPa	,
				AllowGFMEnPa:=emC_PPC[PPCNum].Param.AllowGFMEnPa	,
				BlackSys	:=  emC_PPC[PPCNum].LuC[LuCNum].Out.BlackSys	
				)	;
								
								
									
	L5_FSetOut_Q	:=	emC_PPC_LuCOut_5.FSetOut_Q	;					
	L5_USetOut_Q	:=	emC_PPC_LuCOut_5.USetOut_Q	;					
	L5_PSetOut_Q	:=	emC_PPC_LuCOut_5.PSetOut_Q	;					
	L5_QSetOut_Q	:=	emC_PPC_LuCOut_5.QSetOut_Q	;					
	L5_FastFSetOut_Q	:=	emC_PPC_LuCOut_5.FastFSetOut_Q	;					
	L5_FastUSetOut_Q	:=	emC_PPC_LuCOut_5.FastUSetOut_Q	;					
	L5_FastPSetOut_Q	:=	emC_PPC_LuCOut_5.FastPSetOut_Q	;					
	L5_FastQSetOut_Q	:=	emC_PPC_LuCOut_5.FastQSetOut_Q	;					
	L5_FastF_SF_Q	:=	emC_PPC_LuCOut_5.FastF_SF_Q	;					
	L5_FastU_SF_Q	:=	emC_PPC_LuCOut_5.FastU_SF_Q	;					
	L5_FastP_SF_Q	:=	emC_PPC_LuCOut_5.FastP_SF_Q	;							
	L5_NetOnlineSt_Q	:=	emC_PPC_LuCOut_5.NetOnlineSt_Q	;					
	L5_NetIslandReq_Q	:=	emC_PPC_LuCOut_5.NetIslandReq_Q	;					
	L5_AutoStartCmd_Q	:=	emC_PPC_LuCOut_5.AutoStartCmd_Q	;					
	L5_AutoStopCmd_Q	:=	emC_PPC_LuCOut_5.AutoStopCmd_Q	;
							
						
					
END_PROGRAM

PROGRAM emC_LUC_R01_MSH_In
  VAR
    AllowGFMEnPa_S : BOOL := TRUE;
    FNomPa_S : REAL := 50.0;
    UNomPa_S : REAL := 480.0;
    PQFVSelPaGfm_S : BOOL := FALSE;
    PQFVSelPaGfw_S : BOOL := TRUE;
    InvertHwEnablePa_S : BOOL := FALSE;
    AllowGFWEnPa_S : BOOL := TRUE;
    BatStartingTimePa_S : DINT := 30;
    BatStoppingTimePa_S : DINT := 30;
    CmdOutTimePa_S : DINT := 3;
    CoolingTimePa_S : DINT := 30;
    MinRunTimePa_S : DINT := 30;
    StartingTimePa_S : DINT := 30;
    StoppingTimePa_S : DINT := 30;
    LogDisPa_S : BOOL;
    SchedulerStartStopCmdEnPa_S : BOOL := FALSE;
    StartStopEnablePa_S : BOOL := TRUE;
    PhaseRotationPa_S : BOOL := FALSE;
    PLimMaxPa_S : REAL := 1000.0;
    PLimMinPa_S : REAL := -1000.0;
    QLimMaxPa_S : REAL := 300.0;
    QLimMinPa_S : REAL := -300.0;
    FastSlowDataEnPa_S : BOOL := FALSE;
    Q_StoprampDownPa_S : REAL := 10.0;
    Q_StoprampUpPa_S : REAL := 10.0;
    emC_PPCIn_1 : emC_LuC_PPCIn;
    SetPointRampEnPa_S : BOOL := TRUE;
    PPC_SetPointRampEnPa_S : BOOL := TRUE;
    PPC_FSetOutRmpUpPa_S : REAL := 0.05;
    PPC_FSetOutRmpDownPa_S : REAL := 0.05;
    PPC_USetOutRmpUpPa_S : REAL := 10.0;
    PPC_USetOutRmpDownPa_S : REAL := 10.0;
    PPC_PSetOutRmpUpPa_S : REAL := 10.0;
    PPC_PSetOutRmpDownPa_S : REAL := 10.0;
    PPC_QSetOutRmpUpPa_S : REAL := 10.0;
    PPC_QSetOutRmpDownPa_S : REAL := 10.0;
  END_VAR
  VAR_EXTERNAL
    LUC_Num : INT;
    emC_LUC : emC_LUC_Array;
  END_VAR
  VAR
    PLCMODE_RUN : BOOL;
    BatPlc_MbCommTOutPa_S : DINT := 3;
    BatPlc_MessageTimeDelayPa_S : DINT := 5;
    BatPlc_NbOfRackPa_S : INT := 5;
    BatPlc_NbOfBankPa_S : INT := 1;
    BatPlc_InvDcBusUMinPa_S : REAL := 600.0;
    BatPlc_BattSysSyncUBiasPa_S : REAL := 0.0;
    BatPlc_InvDcBusUMaxPa_S : REAL := 1000.0;
    BatPlc_BattRackNomPActPa_S : REAL := 87.5;
    BatPlc_RacksStartToutPa_S : DINT := 30;
    BatPlc_SYSSyncRangePa_S : REAL := 5.0;
    BatPlc_RacksStopngTimeoutPa_S : DINT := 30;
    BatPlc_EnDerateWrtSocPa_S : BOOL;
    BatPlc_EnDerateWrtTempPa_S : BOOL;
    BatPlc_ClockSyncIntervalPa_S : DINT := 5;
    BatPlc_WatchDogModePa_S : INT;
    BatPlc_ClockSyncEnPA_S : BOOL;
    BatPlc_InvPActMaxPa_S : REAL := 1000.0;
    BatPlc_MinPctOfRkPa_S : REAL := 80.0;
    BatPlc_InvPActMinPa_S : REAL := 0.0;
    BatPlc_BattRackNomEActPa_S : REAL;
    MapOfRackPa_S : MapOfRackStruct;
    S_PRMS_FSO_MNG_1 : S_PRMS_FSO_MNG;
    S_PRMS_FSO_MNG_2 : S_PRMS_FSO_MNG;
    S_PRMS_FSO_MNG_3 : S_PRMS_FSO_MNG;
    S_PRMS_FSO_MNG_4 : S_PRMS_FSO_MNG;
    Timestamp : Timestamp;
    FirstRun : BOOL := TRUE;
    QCtrlStopDeadbPa_S : REAL := 10.0;
    PCtrlStopDeadbPa_S : REAL := 10.0;
    P_StoprampUpPa_S : REAL := 10.0;
    P_StoprampDownPa_S : REAL := 10.0;
    S_FSO_MNG_5 : S_FSO_MNG;
    S_PRMS_FSO_MNG_5 : S_PRMS_FSO_MNG;
    SelModMapPa_S : INT := 1;
    BatPlc_DrtChOnSocLUpSocPaPt1_S : REAL := 0.0;
    BatPlc_DrtChOnSocLUpSocPaPt2_S : REAL := 0.0;
    BatPlc_DrtChOnSocLUpSocPaPt3_S : REAL := 0.0;
    BatPlc_DrtChOnSocLUpSocPaPt4_S : REAL;
    BatPlc_DrtChOnSocLUpSocPaPt5_S : REAL;
    BatPlc_DrtChOnSocLUpSocPaPt6_S : REAL;
    BatPlc_DrtChOnSocLUpDrtPaPt1_S : REAL;
    BatPlc_DrtChOnSocLUpDrtPaPt2_S : REAL;
    BatPlc_DrtChOnSocLUpDrtPaPt3_S : REAL;
    BatPlc_DrtChOnSocLUpDrtPaPt4_S : REAL;
    BatPlc_DrtChOnSocLUpDrtPaPt5_S : REAL;
    BatPlc_DrtChOnSocLUpDrtPaPt6_S : REAL;
    BatPlc_DrtDsOnSocLUpSocPaPt1_S : REAL;
    BatPlc_DrtDsOnSocLUpSocPaPt2_S : REAL;
    BatPlc_DrtDsOnSocLUpSocPaPt3_S : REAL;
    BatPlc_DrtDsOnSocLUpSocPaPt4_S : REAL;
    BatPlc_DrtDsOnSocLUpSocPaPt5_S : REAL;
    BatPlc_DrtDsOnSocLUpSocPaPt6_S : REAL;
    BatPlc_DrtDsOnSocLUpDrtPaPt1_S : REAL;
    BatPlc_DrtDsOnSocLUpDrtPaPt2_S : REAL;
    BatPlc_DrtDsOnSocLUpDrtPaPt3_S : REAL;
    BatPlc_DrtDsOnSocLUpDrtPaPt4_S : REAL;
    BatPlc_DrtDsOnSocLUpDrtPaPt5_S : REAL;
    BatPlc_DrtDsOnSocLUpDrtPaPt6_S : REAL;
    BatPlc_DrtTempLUpTempPaPt1_S : REAL;
    BatPlc_DrtTempLUpTempPaPt2_S : REAL;
    BatPlc_DrtTempLUpTempPaPt3_S : REAL;
    BatPlc_DrtTempLUpTempPaPt4_S : REAL;
    BatPlc_DrtTempLUpTempPaPt5_S : REAL;
    BatPlc_DrtTempLUpTempPaPt6_S : REAL;
    BatPlc_DrtTempLUpDeratePaPt1_S : REAL;
    BatPlc_DrtTempLUpDeratePaPt2_S : REAL;
    BatPlc_DrtTempLUpDeratePaPt3_S : REAL;
    BatPlc_DrtTempLUpDeratePaPt4_S : REAL;
    BatPlc_DrtTempLUpDeratePaPt5_S : REAL;
    BatPlc_DrtTempLUpDeratePaPt6_S : REAL;
    Red_S : INT;
    Red : INT;
    S_FSO_MNG_1 : S_FSO_MNG;
    S_FSO_MNG_2 : S_FSO_MNG;
    S_FSO_MNG_3 : S_FSO_MNG;
    S_FSO_MNG_4 : S_FSO_MNG;
    S_SCO_MNG_5 : S_SCO_MNG;
    S_SCO_MNG_6 : S_SCO_MNG;
    S_SCO_MNG_7 : S_SCO_MNG;
    S_SCO_MNG_8 : S_SCO_MNG;
    S_SCO_MNG_9 : S_SCO_MNG;
    FSetOut_Q : FSO;
    USetOut_Q : FSO;
    PSetOut_Q : FSO;
    QSetOut_Q : FSO;
    NetOnlineSt_Q : SCO;
    NetIslandReq_Q : SCO;
    AutoStartCmd_Q : SCO;
    AutoStopCmd_Q : SCO;
    StopRampSt_Q : SCO;
    FSetOut_I : FSO;
    USetOut_I : FSO;
    PSetOut_I : FSO;
    QSetOut_I : FSO;
    NetOnlineSt_I : SCO;
    NetIslandReq_I : SCO;
    AutoStartCmd_I : SCO;
    AutoStopCmd_I : SCO;
    StopRampSt_I : SCO;
    StartCmd_I : SCO;
    StopCmd_I : SCO;
    AlarmReset_I : SCO;
    BlackOutResCmd_I : SCO;
    StartCmd_Q : SCO;
    StopCmd_Q : SCO;
    AlarmReset_Q : SCO;
    BlackOutResCmd_Q : SCO;
    S_SCO_MNG_1 : S_SCO_MNG;
    S_SCO_MNG_2 : S_SCO_MNG;
    S_SCO_MNG_3 : S_SCO_MNG;
    S_SCO_MNG_4 : S_SCO_MNG;
  END_VAR

						
							LUC_Num := 1;
Red := Red_S;
emC_LUC[LUC_Num].BattPLC.Pa.MbCommTOutPa			:=	DINT_To_Time (BatPlc_MbCommTOutPa_S * DINT#1000);
emC_LUC[LUC_Num].BattPLC.Pa.MessageTimeDelayPa		:= 	DINT_To_Time (BatPlc_MessageTimeDelayPa_S * DINT#1000);
emC_LUC[LUC_Num].BattPLC.Pa.NbOfRackPa				:=	BatPlc_NbOfRackPa_S	;
emC_LUC[LUC_Num].BattPLC.Pa.NbOfBankPa				:=	BatPlc_NbOfBankPa_S	;
emC_LUC[LUC_Num].BattPLC.Pa.InvDcBusUMinPa			:=	BatPlc_InvDcBusUMinPa_S	;
emC_LUC[LUC_Num].BattPLC.Pa.BattSysSyncUBiasPa		:=	BatPlc_BattSysSyncUBiasPa_S	;
emC_LUC[LUC_Num].BattPLC.Pa.InvDcBusUMaxPa			:=	BatPlc_InvDcBusUMaxPa_S	;
emC_LUC[LUC_Num].BattPLC.Pa.BattRackNomEActPa		:=	BatPlc_BattRackNomEActPa_S	;
emC_LUC[LUC_Num].BattPLC.Pa.BattRackNomPActPa		:=	BatPlc_BattRackNomPActPa_S	;
emC_LUC[LUC_Num].BattPLC.Pa.InvPActMinPa			:=	BatPlc_InvPActMinPa_S	;
emC_LUC[LUC_Num].BattPLC.Pa.InvPActMaxPa			:=	BatPlc_InvPActMaxPa_S	;
emC_LUC[LUC_Num].BattPLC.Pa.MinPctOfRkPa			:=	BatPlc_MinPctOfRkPa_S	;
emC_LUC[LUC_Num].BattPLC.Pa.RacksStartingTimeoutPa	:=	DINT_To_Time(BatPlc_RacksStartToutPa_S * DINT#1000);
emC_LUC[LUC_Num].BattPLC.Pa.Batt_SYSSyncRangePa		:=	BatPlc_SYSSyncRangePa_S	;
emC_LUC[LUC_Num].BattPLC.Pa.DrtChrgOnSocLookUpSocPa[1]	:=	BatPlc_DrtChOnSocLUpSocPaPt1_S	;
emC_LUC[LUC_Num].BattPLC.Pa.DrtChrgOnSocLookUpSocPa[2]	:=	BatPlc_DrtChOnSocLUpSocPaPt2_S	;
emC_LUC[LUC_Num].BattPLC.Pa.DrtChrgOnSocLookUpSocPa[3]	:=	BatPlc_DrtChOnSocLUpSocPaPt3_S	;
emC_LUC[LUC_Num].BattPLC.Pa.DrtChrgOnSocLookUpSocPa[4]	:=	BatPlc_DrtChOnSocLUpSocPaPt4_S	;
emC_LUC[LUC_Num].BattPLC.Pa.DrtChrgOnSocLookUpSocPa[5]	:=	BatPlc_DrtChOnSocLUpSocPaPt5_S	;
emC_LUC[LUC_Num].BattPLC.Pa.DrtChrgOnSocLookUpSocPa[6]	:=	BatPlc_DrtChOnSocLUpSocPaPt6_S	;
								
emC_LUC[LUC_Num].BattPLC.Pa.DrtChrgOnSocLookUpDrtPa[1]	:=	BatPlc_DrtChOnSocLUpDrtPaPt1_S	;
emC_LUC[LUC_Num].BattPLC.Pa.DrtChrgOnSocLookUpDrtPa[2]	:=	BatPlc_DrtChOnSocLUpDrtPaPt2_S	;
emC_LUC[LUC_Num].BattPLC.Pa.DrtChrgOnSocLookUpDrtPa[3]	:=	BatPlc_DrtChOnSocLUpDrtPaPt3_S	;
emC_LUC[LUC_Num].BattPLC.Pa.DrtChrgOnSocLookUpDrtPa[4]	:=	BatPlc_DrtChOnSocLUpDrtPaPt4_S	;
emC_LUC[LUC_Num].BattPLC.Pa.DrtChrgOnSocLookUpDrtPa[5]	:=	BatPlc_DrtChOnSocLUpDrtPaPt5_S	;
emC_LUC[LUC_Num].BattPLC.Pa.DrtChrgOnSocLookUpDrtPa[6]	:=	BatPlc_DrtChOnSocLUpDrtPaPt6_S	;
								
emC_LUC[LUC_Num].BattPLC.Pa.DrtDChrgOnSocLookUpSocPa[1]:=	BatPlc_DrtDsOnSocLUpSocPaPt1_S	;
emC_LUC[LUC_Num].BattPLC.Pa.DrtDChrgOnSocLookUpSocPa[2]:=	BatPlc_DrtDsOnSocLUpSocPaPt2_S	;
emC_LUC[LUC_Num].BattPLC.Pa.DrtDChrgOnSocLookUpSocPa[3]:=	BatPlc_DrtDsOnSocLUpSocPaPt3_S	;
emC_LUC[LUC_Num].BattPLC.Pa.DrtDChrgOnSocLookUpSocPa[4]:=	BatPlc_DrtDsOnSocLUpSocPaPt4_S	;
emC_LUC[LUC_Num].BattPLC.Pa.DrtDChrgOnSocLookUpSocPa[5]:=	BatPlc_DrtDsOnSocLUpSocPaPt5_S	;
emC_LUC[LUC_Num].BattPLC.Pa.DrtDChrgOnSocLookUpSocPa[6]:=	BatPlc_DrtDsOnSocLUpSocPaPt6_S	;
								
emC_LUC[LUC_Num].BattPLC.Pa.DrtDChrgOnSocLookUpDrtPa[1]:=	BatPlc_DrtDsOnSocLUpDrtPaPt1_S	;
emC_LUC[LUC_Num].BattPLC.Pa.DrtDChrgOnSocLookUpDrtPa[2]:=	BatPlc_DrtDsOnSocLUpDrtPaPt2_S	;
emC_LUC[LUC_Num].BattPLC.Pa.DrtDChrgOnSocLookUpDrtPa[3]:=	BatPlc_DrtDsOnSocLUpDrtPaPt3_S	;
emC_LUC[LUC_Num].BattPLC.Pa.DrtDChrgOnSocLookUpDrtPa[4]:=	BatPlc_DrtDsOnSocLUpDrtPaPt4_S	;
emC_LUC[LUC_Num].BattPLC.Pa.DrtDChrgOnSocLookUpDrtPa[5]:=	BatPlc_DrtDsOnSocLUpDrtPaPt5_S	;
emC_LUC[LUC_Num].BattPLC.Pa.DrtDChrgOnSocLookUpDrtPa[6]:=	BatPlc_DrtDsOnSocLUpDrtPaPt6_S	;
								
emC_LUC[LUC_Num].BattPLC.Pa.DerateTempLookUpTempPa[1]	:=	BatPlc_DrtTempLUpTempPaPt1_S	;
emC_LUC[LUC_Num].BattPLC.Pa.DerateTempLookUpTempPa[2]	:=	BatPlc_DrtTempLUpTempPaPt2_S	;
emC_LUC[LUC_Num].BattPLC.Pa.DerateTempLookUpTempPa[3]	:=	BatPlc_DrtTempLUpTempPaPt3_S	;
emC_LUC[LUC_Num].BattPLC.Pa.DerateTempLookUpTempPa[4]	:=	BatPlc_DrtTempLUpTempPaPt4_S	;
emC_LUC[LUC_Num].BattPLC.Pa.DerateTempLookUpTempPa[5]	:=	BatPlc_DrtTempLUpTempPaPt5_S	;
emC_LUC[LUC_Num].BattPLC.Pa.DerateTempLookUpTempPa[6]	:=	BatPlc_DrtTempLUpTempPaPt6_S	;
								
emC_LUC[LUC_Num].BattPLC.Pa.DerateTempLookUpDeratePa[1]	:=	BatPlc_DrtTempLUpDeratePaPt1_S	;
emC_LUC[LUC_Num].BattPLC.Pa.DerateTempLookUpDeratePa[2]	:=	BatPlc_DrtTempLUpDeratePaPt2_S	;
emC_LUC[LUC_Num].BattPLC.Pa.DerateTempLookUpDeratePa[3]	:=	BatPlc_DrtTempLUpDeratePaPt3_S	;
emC_LUC[LUC_Num].BattPLC.Pa.DerateTempLookUpDeratePa[4]	:=	BatPlc_DrtTempLUpDeratePaPt4_S	;
emC_LUC[LUC_Num].BattPLC.Pa.DerateTempLookUpDeratePa[5]	:=	BatPlc_DrtTempLUpDeratePaPt5_S	;
emC_LUC[LUC_Num].BattPLC.Pa.DerateTempLookUpDeratePa[6]	:=	BatPlc_DrtTempLUpDeratePaPt6_S	;
								
								
emC_LUC[LUC_Num].BattPLC.Pa.RacksStoppingTimeoutPa	:=	DINT_TO_TIME(BatPlc_RacksStopngTimeoutPa_S * DINT#1000)	;
emC_LUC[LUC_Num].BattPLC.Pa.EnDerateWrtSocPa		:=	BatPlc_EnDerateWrtSocPa_S	;
emC_LUC[LUC_Num].BattPLC.Pa.EnDerateWrtTempPa		:=	BatPlc_EnDerateWrtTempPa_S	;
emC_LUC[LUC_Num].BattPLC.Pa.ClockSyncIntervalPa		:=	DINT_TO_TIME(BatPlc_ClockSyncIntervalPa_S * DINT#1000)	;
emC_LUC[LUC_Num].BattPLC.Pa.WatchDogModePa			:=	BatPlc_WatchDogModePa_S		;
emC_LUC[LUC_Num].BattPLC.Pa.ClockSyncEnPA			:=	BatPlc_ClockSyncEnPA_S	;
								
(*emPSPArams*)
								
emC_LUC[LUC_Num].emPs.emPsOut.In.AllowGFMEnPa 			:= AllowGFMEnPa_S;
emC_LUC[LUC_Num].emPs.emPsOut.In.AllowGFWEnPa 			:= AllowGFWEnPa_S;
emC_LUC[LUC_Num].emPs.emPsOut.In.FNomPa					:= FNomPa_S;
emC_LUC[LUC_Num].emPs.emPsOut.In.UNomPa	 				:= UNomPa_S;
emC_LUC[LUC_Num].emPs.emPsOut.In.PQFVSelPaGfm	 		:= PQFVSelPaGfm_S;
emC_LUC[LUC_Num].emPs.emPsOut.In.PQFVSelPaGfw	 		:= PQFVSelPaGfw_S;
emC_LUC[LUC_Num].emPs.emPsOut.In.InvertHwEnablePa	 	:= InvertHwEnablePa_S;
emC_LUC[LUC_Num].emPs.emPsOut.In.PhaseRotationPa	 	:= PhaseRotationPa_S;
emC_LUC[LUC_Num].emPs.emPsOut.In.PLimMaxPa	 			:= PLimMaxPa_S;
emC_LUC[LUC_Num].emPs.emPsOut.In.PLimMinPa			 	:= PLimMinPa_S;
emC_LUC[LUC_Num].emPs.emPsOut.In.QLimMaxPa			 	:= QLimMaxPa_S;
emC_LUC[LUC_Num].emPs.emPsOut.In.QLimMinPa			 	:= QLimMinPa_S;
emC_LUC[LUC_Num].emPs.emPsOut.In.FastSlowDataEnPa 		:= FastSlowDataEnPa_S;
emC_LUC[LUC_Num].emPs.emPsOut.In.AllowGFMEnPa 			:= AllowGFMEnPa_S;
emC_LUC[LUC_Num].emPs.emPsOut.In.SelModMapPa			:= SelModMapPa_S;
(*State Machine*)
emC_LUC[LUC_Num].SM.In.BatStartingTimePa 				:= DINT_TO_TIME(BatStartingTimePa_S * DINT#1000);
emC_LUC[LUC_Num].SM.In.BatStoppingTimePa 				:= DINT_TO_TIME(BatStoppingTimePa_S * DINT#1000);
emC_LUC[LUC_Num].SM.In.CmdOutTimePa 					:= DINT_TO_TIME(CmdOutTimePa_S * DINT#1000);
emC_LUC[LUC_Num].SM.In.CoolingTimePa 					:= DINT_TO_TIME(CoolingTimePa_S * DINT#1000);
emC_LUC[LUC_Num].SM.In.LogDisPa 						:= LogDisPa_S;
emC_LUC[LUC_Num].SM.In.MinRunTimePa 					:= DINT_TO_TIME(MinRunTimePa_S * DINT#1000);
emC_LUC[LUC_Num].SM.In.SchedulerStartStopCmdEnPa 		:= SchedulerStartStopCmdEnPa_S;
emC_LUC[LUC_Num].SM.In.StartingTimePa 					:= DINT_TO_TIME(StartingTimePa_S * DINT#1000);
emC_LUC[LUC_Num].SM.In.StartStopEnablePa		 		:=StartStopEnablePa_S;
emC_LUC[LUC_Num].SM.In.StoppingTimePa				 	:= DINT_TO_TIME(StoppingTimePa_S * DINT#1000);
								
(*ControlLibs*)
emC_LUC[LUC_Num].emC_LUC_Ctrl.LUC_BESS_Parameters.P_StoprampDownPa 		:= P_StoprampDownPa_S;
emC_LUC[LUC_Num].emC_LUC_Ctrl.LUC_BESS_Parameters.P_StoprampUpPa 		:= P_StoprampUpPa_S;
emC_LUC[LUC_Num].emC_LUC_Ctrl.LUC_BESS_Parameters.PCtrlDeadbPa 			:= PCtrlStopDeadbPa_S;
emC_LUC[LUC_Num].emC_LUC_Ctrl.LUC_BESS_Parameters.PLimMaxPa 	 		:= 	PLimMaxPa_S;
emC_LUC[LUC_Num].emC_LUC_Ctrl.LUC_BESS_Parameters.PLimMinPa			 	:= 	PLimMinPa_S;
emC_LUC[LUC_Num].emC_LUC_Ctrl.LUC_BESS_Parameters.Q_StoprampDownPa		:= 	Q_StoprampDownPa_S;
emC_LUC[LUC_Num].emC_LUC_Ctrl.LUC_BESS_Parameters.Q_StoprampUpPa		:= 	Q_StoprampUpPa_S;
emC_LUC[LUC_Num].emC_LUC_Ctrl.LUC_BESS_Parameters.QCtrlDeadbPa			:=	QCtrlStopDeadbPa_S;
emC_LUC[LUC_Num].emC_LUC_Ctrl.LUC_BESS_Parameters.QLimMaxPa			 	:= 	QLimMaxPa_S;
emC_LUC[LUC_Num].emC_LUC_Ctrl.LUC_BESS_Parameters.QLimMinPa			 	:= 	QLimMinPa_S;
								
(*PPC Interface*)
emC_LUC[LUC_Num].PPC.PPCIn.In.SetPointRampEnPa					:= PPC_SetPointRampEnPa_S;
emC_LUC[LUC_Num].PPC.PPCIn.In.FSetOutRmpUpPa					:= PPC_FSetOutRmpUpPa_S;
emC_LUC[LUC_Num].PPC.PPCIn.In.FSetOutRmpDownPa					:= PPC_FSetOutRmpDownPa_S;
emC_LUC[LUC_Num].PPC.PPCIn.In.USetOutRmpUpPa					:= PPC_USetOutRmpUpPa_S;
emC_LUC[LUC_Num].PPC.PPCIn.In.USetOutRmpDownPa					:= PPC_USetOutRmpDownPa_S;
emC_LUC[LUC_Num].PPC.PPCIn.In.PSetOutRmpUpPa					:= PPC_PSetOutRmpUpPa_S;
emC_LUC[LUC_Num].PPC.PPCIn.In.PSetOutRmpDownPa					:= PPC_PSetOutRmpDownPa_S;
emC_LUC[LUC_Num].PPC.PPCIn.In.QSetOutRmpUpPa					:= PPC_QSetOutRmpUpPa_S;
emC_LUC[LUC_Num].PPC.PPCIn.In.QSetOutRmpDownPa					:= PPC_QSetOutRmpDownPa_S;
							
							emC_LUC[LUC_Num].Field.MSHIn.ManualSt				:= FALSE;
emC_LUC[LUC_Num].Field.MSHIn.Warning				:= FALSE;
emC_LUC[LUC_Num].Field.MSHIn.NonCriticalAlarm		:= FALSE;
emC_LUC[LUC_Num].Field.MSHIn.CriticalAlarm			:= FALSE;
							
							S_SCO_MNG_1	(ExtCmd_Input_I:=	StartCmd_I	,Cfg_t_delay:=T#1s,Cfg_disCMD:= FALSE);	StartCmd_Q	:=	S_SCO_MNG_1.ExtCmd_Output_Q	;	emC_LUC[LUC_Num].SCADA.In.StartCmd	:=	S_SCO_MNG_1.SCO_Execute_Out	;
S_SCO_MNG_2	(ExtCmd_Input_I:=	StopCmd_I	,Cfg_t_delay:=T#1s,Cfg_disCMD:= FALSE);	StopCmd_Q	:=	S_SCO_MNG_2.ExtCmd_Output_Q	;	emC_LUC[LUC_Num].SCADA.In.StopCmd	:=	S_SCO_MNG_2.SCO_Execute_Out	;
S_SCO_MNG_3	(ExtCmd_Input_I:=	AlarmReset_I	,Cfg_t_delay:=T#1s,Cfg_disCMD:= FALSE);	AlarmReset_Q	:=	S_SCO_MNG_3.ExtCmd_Output_Q	;	emC_LUC[LUC_Num].SCADA.In.AlarmReset	:=	S_SCO_MNG_3.SCO_Execute_Out	;
S_SCO_MNG_4	(ExtCmd_Input_I:=	BlackOutResCmd_I	,Cfg_t_delay:=T#1s,Cfg_disCMD:= FALSE);	BlackOutResCmd_Q	:=	S_SCO_MNG_4.ExtCmd_Output_Q	;	emC_LUC[LUC_Num].SCADA.In.BlackOutResCmd	:=	S_SCO_MNG_4.SCO_Execute_Out	;
								
emC_LUC[LUC_Num].SM.In.OpStartCmd	:=	emC_LUC[LUC_Num].SCADA.In.StartCmd	;
emC_LUC[LUC_Num].SM.In.OpStopCmd	:=	emC_LUC[LUC_Num].SCADA.In.StopCmd	;
emC_LUC[LUC_Num].SM.In.ResetCmd 	:=	emC_LUC[LUC_Num].SCADA.In.AlarmReset	;
							
							
								
emC_PPCIn_1(
	SetPointRampEnPa	:=	emC_LUC[LUC_Num].PPC.PPCIn.In.SetPointRampEnPa	, 		
	FSetOutRmpUpPa	:=	emC_LUC[LUC_Num].PPC.PPCIn.In.FSetOutRmpUpPa	, 		
	FSetOutRmpDownPa	:=	emC_LUC[LUC_Num].PPC.PPCIn.In.FSetOutRmpDownPa	, 			
	USetOutRmpUpPa	:=	emC_LUC[LUC_Num].PPC.PPCIn.In.USetOutRmpUpPa	, 		
	USetOutRmpDownPa	:=	emC_LUC[LUC_Num].PPC.PPCIn.In.USetOutRmpDownPa	, 		
	PSetOutRmpUpPa	:=	emC_LUC[LUC_Num].PPC.PPCIn.In.PSetOutRmpUpPa	, 		
	PSetOutRmpDownPa	:=	emC_LUC[LUC_Num].PPC.PPCIn.In.PSetOutRmpDownPa	, 		
	QSetOutRmpUpPa	:=	emC_LUC[LUC_Num].PPC.PPCIn.In.QSetOutRmpUpPa	,		
	QSetOutRmpDownPa	:=	emC_LUC[LUC_Num].PPC.PPCIn.In.QSetOutRmpDownPa	, 		
					
	PSetOut_I	:=	PSetOut_I	,
	UNomPa	:=	emC_LUC[LUC_Num].emPs.emPsOut.In.UNomPa	,
	FNomPa	:=	emC_LUC[LUC_Num].emPs.emPsOut.In.FNomPa	,
	FastSlowDataEnPa	:=	emC_LUC[LUC_Num].emPs.emPsOut.In.FastSlowDataEnPa	,
	FSetOut_I	:=	FSetOut_I	,
	USetOut_I	:=	USetOut_I	,
	QSetOut_I	:=	QSetOut_I	,
	AutoStopCmd_I	:=	AutoStopCmd_I	,
	AutoStartCmd_I	:=	AutoStartCmd_I	,
	NetOnlineSt_I	:=	NetOnlineSt_I	,
	NetIslandReq_I	:=	NetIslandReq_I	);
								
FSetOut_Q	:=	emC_PPCIn_1.FSetOut_Q	;
USetOut_Q	:=	emC_PPCIn_1.USetOut_Q	;
PSetOut_Q	:=	emC_PPCIn_1.PSetOut_Q	;
QSetOut_Q	:=	emC_PPCIn_1.QSetOut_Q	;
AutoStartCmd_Q	:=	emC_PPCIn_1.AutoStartCmd_Q	;
AutoStopCmd_Q	:=	emC_PPCIn_1.AutoStopCmd_Q	;
NetOnlineSt_Q	:=	emC_PPCIn_1.NetOnlineSt_Q	;
NetIslandReq_Q	:=	emC_PPCIn_1.NetIslandReq_Q	;
emC_LUC[LUC_Num].PPC.PPCIn.Out.USetOut 	:=	emC_PPCIn_1.USetOut	;
emC_LUC[LUC_Num].PPC.PPCIn.Out.FSetOut	:=	emC_PPCIn_1.FSetOut	;
emC_LUC[LUC_Num].PPC.PPCIn.Out.PSetOut	:=	emC_PPCIn_1.PSetOut	;
emC_LUC[LUC_Num].PPC.PPCIn.Out.QSetOut	:=	emC_PPCIn_1.QSetOut	;
emC_LUC[LUC_Num].PPC.PPCIn.Out.AutoStartCmd	:=	emC_PPCIn_1.AutoStartCmd	;
emC_LUC[LUC_Num].PPC.PPCIn.Out.AutoStopCmd	:=	emC_PPCIn_1.AutoStopCmd	;
emC_LUC[LUC_Num].PPC.PPCIn.Out.NetOnlineSt	:=	emC_PPCIn_1.NetOnlineSt	;
emC_LUC[LUC_Num].PPC.PPCIn.Out.NetIslandReq	:=	emC_PPCIn_1.NetIslandReq	;
							
						
					
END_PROGRAM

PROGRAM emC_LUC_R02_DevIn
  VAR
    StVnd_I : MFI;
    PPVphAB_I : MFI;
    PPVphBC_I : MFI;
    PPVphCA_I : MFI;
    PhVphA_I : MFI;
    PhVphB_I : MFI;
    PhVphC_I : MFI;
    V_SF_I : MFI;
    W_I : MFI;
    W_SF_I : MFI;
    Hz_I : MFI;
    Hz_SF_I : MFI;
    VA_I : MFI;
    VA_SF_I : MFI;
    RVAr_I : MFI;
    VAr_SF_I : MFI;
    Pf_I : MFI;
    PF_SF_I : MFI;
    WH_I : MFI;
    WH_SF_I : MFI;
    PSR_R_CMD_I : TDC;
    PSR2_R_CMD_I : TDC;
    emC_E_StateMachine_1 : emC_E_StateMachine;
    TON_5 : TON;
    Timestamp_To_String_1 : Timestamp_To_String;
    Bmsrack : BMS_RackArray;
    bmssys : BMS_Sys;
    MbOut : MbCtrlStruct;
    emC_BatPlcParameters_1 : emC_BatPlcParameters;
    emC_BatMBus_SDI_V_1_1_10_1 : emC_BatMBus_SDI_V_1_1_10;
    emC_BatPLCLogic_1 : emC_BatPLCLogic;
    BattPLCCmd_Resp_I : TDC;
    BatPLC_TDC_Resp_I : TDC;
    BatPLC_TDC_Req_Q : TDC;
    emPS_In_1 : emPS_In;
    A_SF_I : MFI;
    A_I : MFI;
    AphA_I : MFI;
    AphB_I : MFI;
    AphC_I : MFI;
  END_VAR
  VAR_EXTERNAL
    LUC_Num : INT;
    emC_LUC : emC_LUC_Array;
    PLCMODE_RUN : BOOL;
  END_VAR
  VAR
    Sim_On_Pa : BOOL := False;
    Sim_Stop : REAL;
    TON_1 : TON;
    pippo : TDC;
    BattPLCCmd_Req_I : TDC;
    BattPLCCmd_Req_Q : TDC;
    BattPLCCmd2_Req_Q : TDC;
    BattPLCCmd2_Req_I : TDC;
    ForceWrite : BOOL;
  END_VAR

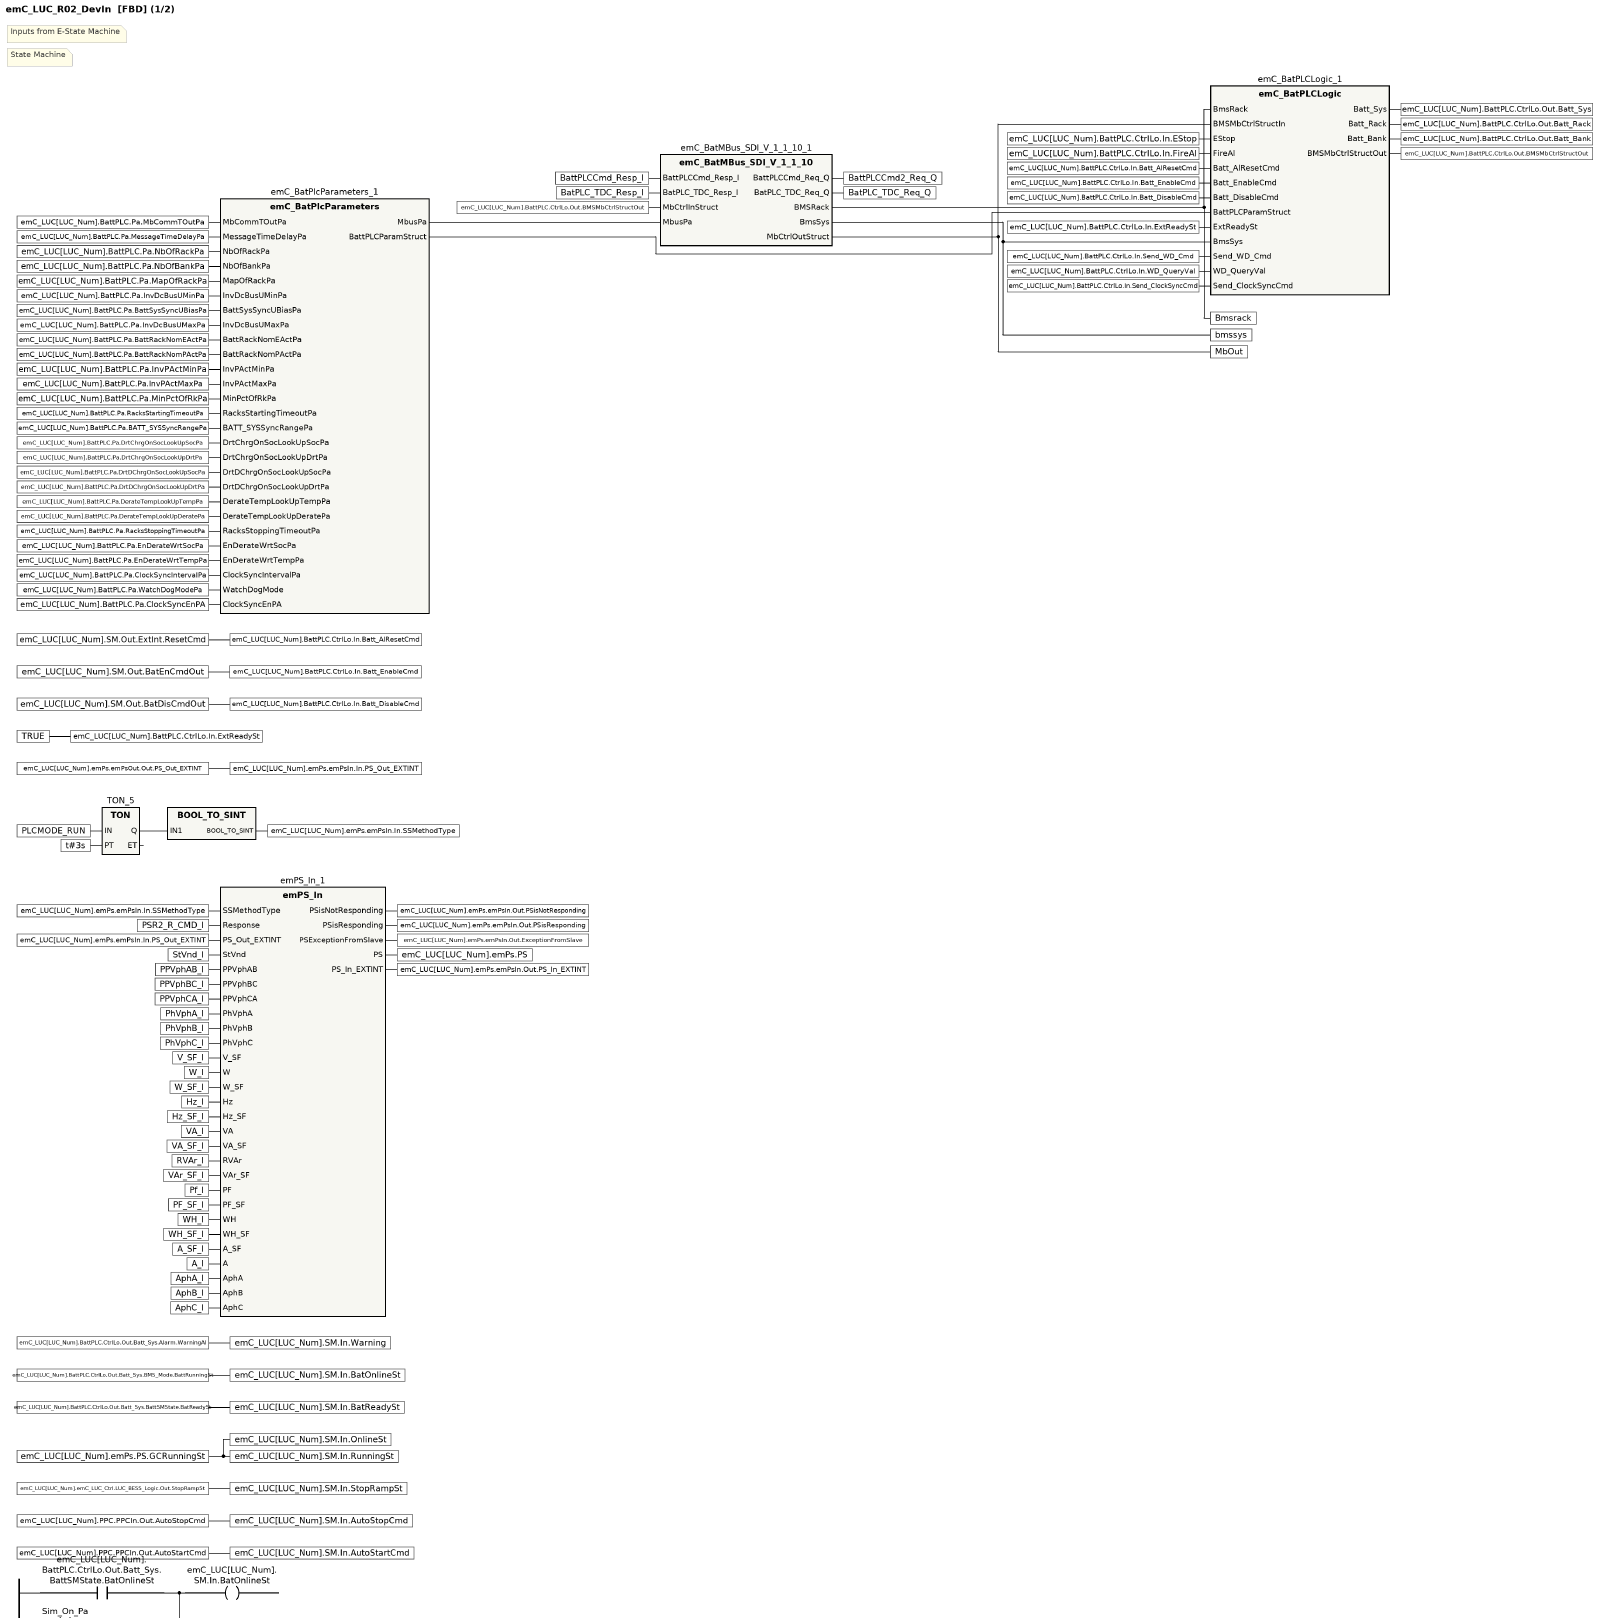
(* FBD diagram, written out as Structured Text *)
(* Inputs from E-State Machine *)
emC_LUC[LUC_Num].BattPLC.CtrlLo.In.Batt_EnableCmd := emC_LUC[LUC_Num].SM.Out.BatEnCmdOut;
emC_LUC[LUC_Num].BattPLC.CtrlLo.In.Batt_DisableCmd := emC_LUC[LUC_Num].SM.Out.BatDisCmdOut;
emC_LUC[LUC_Num].BattPLC.CtrlLo.In.Batt_AlResetCmd := emC_LUC[LUC_Num].SM.Out.ExtInt.ResetCmd;
emC_LUC[LUC_Num].BattPLC.CtrlLo.In.ExtReadySt := TRUE;
emC_BatPlcParameters_1(MbCommTOutPa := emC_LUC[LUC_Num].BattPLC.Pa.MbCommTOutPa, MessageTimeDelayPa := emC_LUC[LUC_Num].BattPLC.Pa.MessageTimeDelayPa, NbOfRackPa := emC_LUC[LUC_Num].BattPLC.Pa.NbOfRackPa, NbOfBankPa := emC_LUC[LUC_Num].BattPLC.Pa.NbOfBankPa, MapOfRackPa := emC_LUC[LUC_Num].BattPLC.Pa.MapOfRackPa, InvDcBusUMinPa := emC_LUC[LUC_Num].BattPLC.Pa.InvDcBusUMinPa, BattSysSyncUBiasPa := emC_LUC[LUC_Num].BattPLC.Pa.BattSysSyncUBiasPa, InvDcBusUMaxPa := emC_LUC[LUC_Num].BattPLC.Pa.InvDcBusUMaxPa, BattRackNomEActPa := emC_LUC[LUC_Num].BattPLC.Pa.BattRackNomEActPa, BattRackNomPActPa := emC_LUC[LUC_Num].BattPLC.Pa.BattRackNomPActPa, InvPActMinPa := emC_LUC[LUC_Num].BattPLC.Pa.InvPActMinPa, InvPActMaxPa := emC_LUC[LUC_Num].BattPLC.Pa.InvPActMaxPa, MinPctOfRkPa := emC_LUC[LUC_Num].BattPLC.Pa.MinPctOfRkPa, RacksStartingTimeoutPa := emC_LUC[LUC_Num].BattPLC.Pa.RacksStartingTimeoutPa, BATT_SYSSyncRangePa := emC_LUC[LUC_Num].BattPLC.Pa.BATT_SYSSyncRangePa, DrtChrgOnSocLookUpSocPa := emC_LUC[LUC_Num].BattPLC.Pa.DrtChrgOnSocLookUpSocPa, DrtChrgOnSocLookUpDrtPa := emC_LUC[LUC_Num].BattPLC.Pa.DrtChrgOnSocLookUpDrtPa, DrtDChrgOnSocLookUpSocPa := emC_LUC[LUC_Num].BattPLC.Pa.DrtDChrgOnSocLookUpSocPa, DrtDChrgOnSocLookUpDrtPa := emC_LUC[LUC_Num].BattPLC.Pa.DrtDChrgOnSocLookUpDrtPa, DerateTempLookUpTempPa := emC_LUC[LUC_Num].BattPLC.Pa.DerateTempLookUpTempPa, DerateTempLookUpDeratePa := emC_LUC[LUC_Num].BattPLC.Pa.DerateTempLookUpDeratePa, RacksStoppingTimeoutPa := emC_LUC[LUC_Num].BattPLC.Pa.RacksStoppingTimeoutPa, EnDerateWrtSocPa := emC_LUC[LUC_Num].BattPLC.Pa.EnDerateWrtSocPa, EnDerateWrtTempPa := emC_LUC[LUC_Num].BattPLC.Pa.EnDerateWrtTempPa, ClockSyncIntervalPa := emC_LUC[LUC_Num].BattPLC.Pa.ClockSyncIntervalPa, WatchDogMode := emC_LUC[LUC_Num].BattPLC.Pa.WatchDogModePa, ClockSyncEnPA := emC_LUC[LUC_Num].BattPLC.Pa.ClockSyncEnPA);
emC_BatMBus_SDI_V_1_1_10_1(BattPLCCmd_Resp_I := BattPLCCmd_Resp_I, BatPLC_TDC_Resp_I := BatPLC_TDC_Resp_I, MbCtrlInStruct := emC_LUC[LUC_Num].BattPLC.CtrlLo.Out.BMSMbCtrlStructOut, MbusPa := emC_BatPlcParameters_1.MbusPa);
BattPLCCmd2_Req_Q := emC_BatMBus_SDI_V_1_1_10_1.BattPLCCmd_Req_Q;
BatPLC_TDC_Req_Q := emC_BatMBus_SDI_V_1_1_10_1.BatPLC_TDC_Req_Q;
MbOut := emC_BatMBus_SDI_V_1_1_10_1.MbCtrlOutStruct;
bmssys := emC_BatMBus_SDI_V_1_1_10_1.BmsSys;
Bmsrack := emC_BatMBus_SDI_V_1_1_10_1.BMSRack;
emC_BatPLCLogic_1(BmsRack := emC_BatMBus_SDI_V_1_1_10_1.BMSRack, BMSMbCtrlStructIn := emC_BatMBus_SDI_V_1_1_10_1.MbCtrlOutStruct, EStop := emC_LUC[LUC_Num].BattPLC.CtrlLo.In.EStop, FireAl := emC_LUC[LUC_Num].BattPLC.CtrlLo.In.FireAl, Batt_AlResetCmd := emC_LUC[LUC_Num].BattPLC.CtrlLo.In.Batt_AlResetCmd, Batt_EnableCmd := emC_LUC[LUC_Num].BattPLC.CtrlLo.In.Batt_EnableCmd, Batt_DisableCmd := emC_LUC[LUC_Num].BattPLC.CtrlLo.In.Batt_DisableCmd, BattPLCParamStruct := emC_BatPlcParameters_1.BattPLCParamStruct, ExtReadySt := emC_LUC[LUC_Num].BattPLC.CtrlLo.In.ExtReadySt, BmsSys := emC_BatMBus_SDI_V_1_1_10_1.BmsSys, Send_WD_Cmd := emC_LUC[LUC_Num].BattPLC.CtrlLo.In.Send_WD_Cmd, WD_QueryVal := emC_LUC[LUC_Num].BattPLC.CtrlLo.In.WD_QueryVal, Send_ClockSyncCmd := emC_LUC[LUC_Num].BattPLC.CtrlLo.In.Send_ClockSyncCmd);
emC_LUC[LUC_Num].BattPLC.CtrlLo.Out.Batt_Sys := emC_BatPLCLogic_1.Batt_Sys;
emC_LUC[LUC_Num].BattPLC.CtrlLo.Out.Batt_Rack := emC_BatPLCLogic_1.Batt_Rack;
emC_LUC[LUC_Num].BattPLC.CtrlLo.Out.Batt_Bank := emC_BatPLCLogic_1.Batt_Bank;
emC_LUC[LUC_Num].BattPLC.CtrlLo.Out.BMSMbCtrlStructOut := emC_BatPLCLogic_1.BMSMbCtrlStructOut;
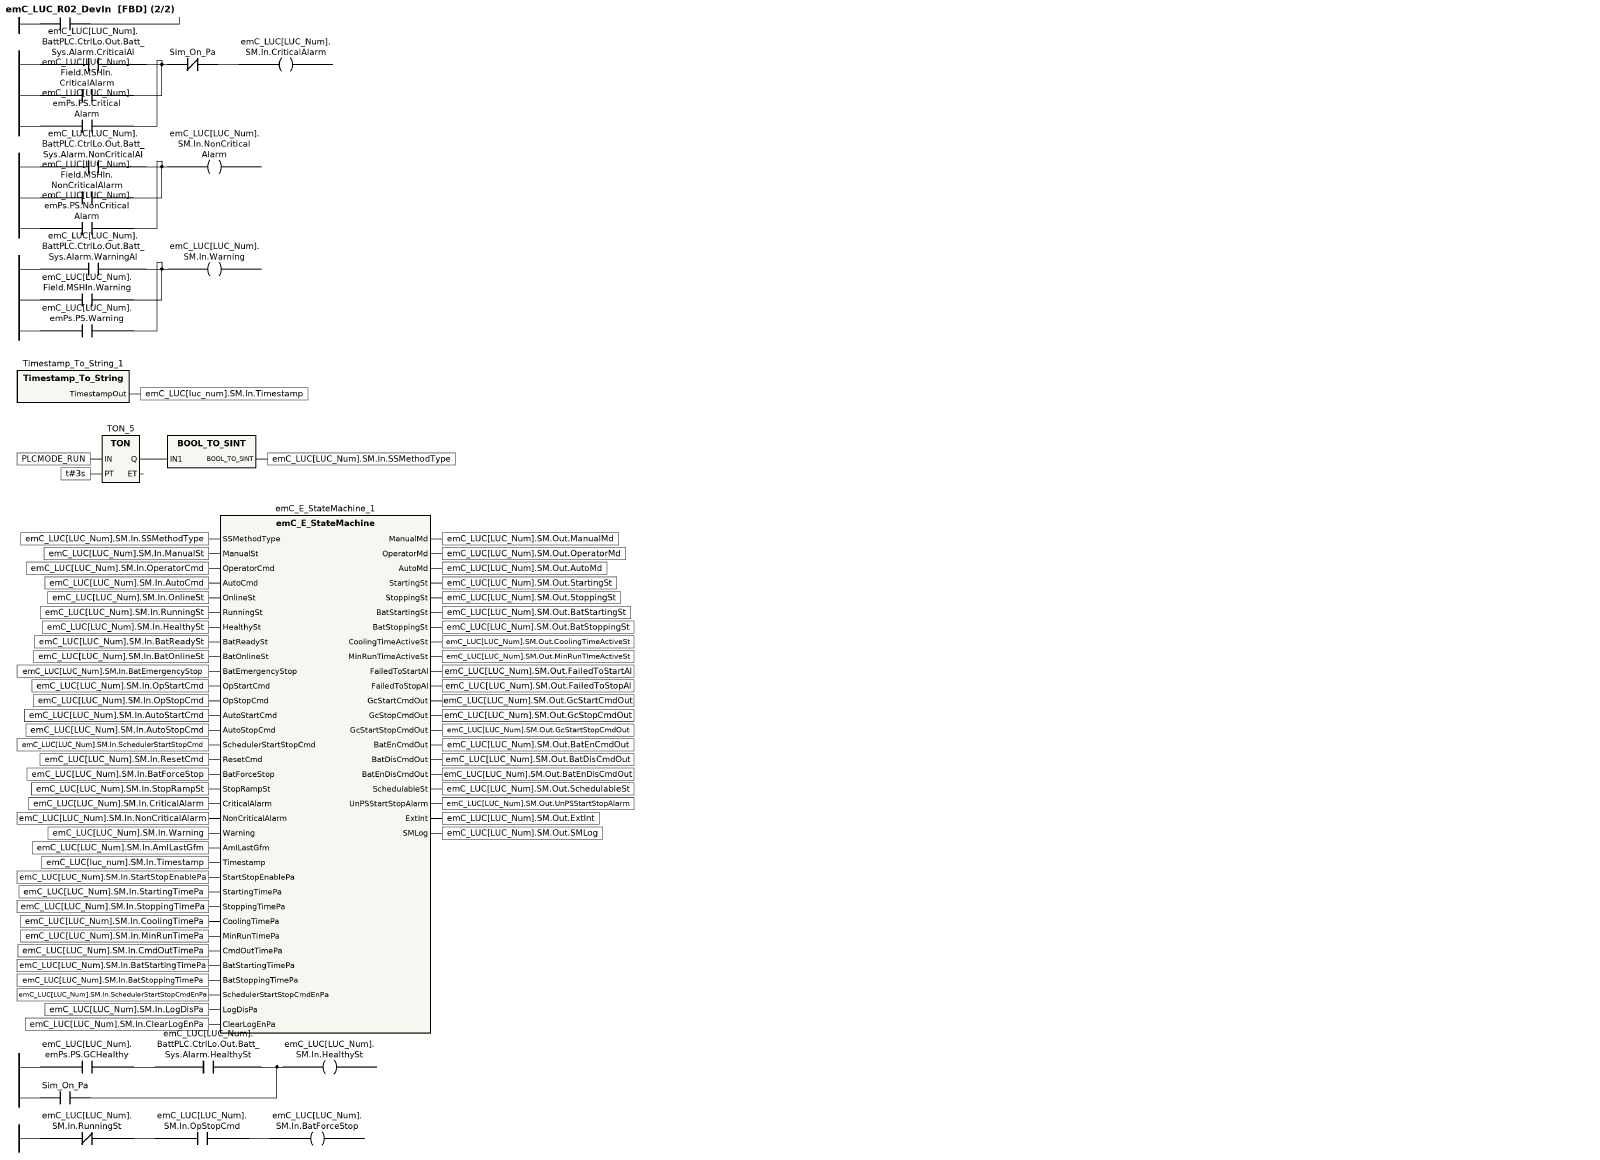
TON_5(IN := PLCMODE_RUN, PT := t#3s);
emC_LUC[LUC_Num].emPs.emPsIn.In.SSMethodType := BOOL_TO_SINT(TON_5.Q);
emC_LUC[LUC_Num].emPs.emPsIn.In.PS_Out_EXTINT := emC_LUC[LUC_Num].emPs.emPsOut.Out.PS_Out_EXTINT;
emPS_In_1(SSMethodType := emC_LUC[LUC_Num].emPs.emPsIn.In.SSMethodType, Response := PSR2_R_CMD_I, PS_Out_EXTINT := emC_LUC[LUC_Num].emPs.emPsIn.In.PS_Out_EXTINT, StVnd := StVnd_I, PPVphAB := PPVphAB_I, PPVphBC := PPVphBC_I, PPVphCA := PPVphCA_I, PhVphA := PhVphA_I, PhVphB := PhVphB_I, PhVphC := PhVphC_I, V_SF := V_SF_I, W := W_I, W_SF := W_SF_I, Hz := Hz_I, Hz_SF := Hz_SF_I, VA := VA_I, VA_SF := VA_SF_I, RVAr := RVAr_I, VAr_SF := VAr_SF_I, PF := Pf_I, PF_SF := PF_SF_I, WH := WH_I, WH_SF := WH_SF_I, A_SF := A_SF_I, A := A_I, AphA := AphA_I, AphB := AphB_I, AphC := AphC_I);
emC_LUC[LUC_Num].emPs.emPsIn.Out.PSisNotResponding := emPS_In_1.PSisNotResponding;
emC_LUC[LUC_Num].emPs.emPsIn.Out.PSisResponding := emPS_In_1.PSisResponding;
emC_LUC[LUC_Num].emPs.emPsIn.Out.ExceptionFromSlave := emPS_In_1.PSExceptionFromSlave;
emC_LUC[LUC_Num].emPs.emPsIn.Out.PS_In_EXTINT := emPS_In_1.PS_In_EXTINT;
emC_LUC[LUC_Num].emPs.PS := emPS_In_1.PS;
(* State Machine *)
TON_5(IN := PLCMODE_RUN, PT := t#3s);
emC_LUC[LUC_Num].SM.In.SSMethodType := BOOL_TO_SINT(TON_5.Q);
Timestamp_To_String_1();
emC_LUC[luc_num].SM.In.Timestamp := Timestamp_To_String_1.TimestampOut;
emC_LUC[LUC_Num].SM.In.CriticalAlarm := (emC_LUC[LUC_Num].BattPLC.CtrlLo.Out.Batt_Sys.Alarm.CriticalAl OR emC_LUC[LUC_Num].Field.MSHIn.CriticalAlarm OR emC_LUC[LUC_Num].emPs.PS.CriticalAlarm) AND NOT Sim_On_Pa;
emC_LUC[LUC_Num].SM.In.NonCriticalAlarm := emC_LUC[LUC_Num].BattPLC.CtrlLo.Out.Batt_Sys.Alarm.NonCriticalAl OR emC_LUC[LUC_Num].Field.MSHIn.NonCriticalAlarm OR emC_LUC[LUC_Num].emPs.PS.NonCriticalAlarm;
emC_LUC[LUC_Num].SM.In.Warning := emC_LUC[LUC_Num].BattPLC.CtrlLo.Out.Batt_Sys.Alarm.WarningAl OR emC_LUC[LUC_Num].Field.MSHIn.Warning OR emC_LUC[LUC_Num].emPs.PS.Warning;
emC_LUC[LUC_Num].SM.In.Warning := emC_LUC[LUC_Num].BattPLC.CtrlLo.Out.Batt_Sys.Alarm.WarningAl;
emC_LUC[LUC_Num].SM.In.BatOnlineSt := emC_LUC[LUC_Num].BattPLC.CtrlLo.Out.Batt_Sys.BMS_Mode.BattRunningSt;
emC_LUC[LUC_Num].SM.In.BatOnlineSt := emC_LUC[LUC_Num].BattPLC.CtrlLo.Out.Batt_Sys.BattSMState.BatOnlineSt OR Sim_On_Pa;
emC_LUC[LUC_Num].SM.In.BatReadySt := emC_LUC[LUC_Num].BattPLC.CtrlLo.Out.Batt_Sys.BattSMState.BatReadySt;
emC_LUC[LUC_Num].SM.In.HealthySt := Sim_On_Pa OR emC_LUC[LUC_Num].emPs.PS.GCHealthy AND emC_LUC[LUC_Num].BattPLC.CtrlLo.Out.Batt_Sys.Alarm.HealthySt;
emC_LUC[LUC_Num].SM.In.OnlineSt := emC_LUC[LUC_Num].emPs.PS.GCRunningSt;
emC_LUC[LUC_Num].SM.In.RunningSt := emC_LUC[LUC_Num].emPs.PS.GCRunningSt;
emC_LUC[LUC_Num].SM.In.StopRampSt := emC_LUC[LUC_Num].emC_LUC_Ctrl.LUC_BESS_Logic.Out.StopRampSt;
emC_LUC[LUC_Num].SM.In.AutoStopCmd := emC_LUC[LUC_Num].PPC.PPCIn.Out.AutoStopCmd;
emC_LUC[LUC_Num].SM.In.AutoStartCmd := emC_LUC[LUC_Num].PPC.PPCIn.Out.AutoStartCmd;
emC_LUC[LUC_Num].SM.In.BatForceStop := NOT emC_LUC[LUC_Num].SM.In.RunningSt AND emC_LUC[LUC_Num].SM.In.OpStopCmd;
emC_E_StateMachine_1(SSMethodType := emC_LUC[LUC_Num].SM.In.SSMethodType, ManualSt := emC_LUC[LUC_Num].SM.In.ManualSt, OperatorCmd := emC_LUC[LUC_Num].SM.In.OperatorCmd, AutoCmd := emC_LUC[LUC_Num].SM.In.AutoCmd, OnlineSt := emC_LUC[LUC_Num].SM.In.OnlineSt, RunningSt := emC_LUC[LUC_Num].SM.In.RunningSt, HealthySt := emC_LUC[LUC_Num].SM.In.HealthySt, BatReadySt := emC_LUC[LUC_Num].SM.In.BatReadySt, BatOnlineSt := emC_LUC[LUC_Num].SM.In.BatOnlineSt, BatEmergencyStop := emC_LUC[LUC_Num].SM.In.BatEmergencyStop, OpStartCmd := emC_LUC[LUC_Num].SM.In.OpStartCmd, OpStopCmd := emC_LUC[LUC_Num].SM.In.OpStopCmd, AutoStartCmd := emC_LUC[LUC_Num].SM.In.AutoStartCmd, AutoStopCmd := emC_LUC[LUC_Num].SM.In.AutoStopCmd, SchedulerStartStopCmd := emC_LUC[LUC_Num].SM.In.SchedulerStartStopCmd, ResetCmd := emC_LUC[LUC_Num].SM.In.ResetCmd, BatForceStop := emC_LUC[LUC_Num].SM.In.BatForceStop, StopRampSt := emC_LUC[LUC_Num].SM.In.StopRampSt, CriticalAlarm := emC_LUC[LUC_Num].SM.In.CriticalAlarm, NonCriticalAlarm := emC_LUC[LUC_Num].SM.In.NonCriticalAlarm, Warning := emC_LUC[LUC_Num].SM.In.Warning, AmILastGfm := emC_LUC[LUC_Num].SM.In.AmILastGfm, Timestamp := emC_LUC[luc_num].SM.In.Timestamp, StartStopEnablePa := emC_LUC[LUC_Num].SM.In.StartStopEnablePa, StartingTimePa := emC_LUC[LUC_Num].SM.In.StartingTimePa, StoppingTimePa := emC_LUC[LUC_Num].SM.In.StoppingTimePa, CoolingTimePa := emC_LUC[LUC_Num].SM.In.CoolingTimePa, MinRunTimePa := emC_LUC[LUC_Num].SM.In.MinRunTimePa, CmdOutTimePa := emC_LUC[LUC_Num].SM.In.CmdOutTimePa, BatStartingTimePa := emC_LUC[LUC_Num].SM.In.BatStartingTimePa, BatStoppingTimePa := emC_LUC[LUC_Num].SM.In.BatStoppingTimePa, SchedulerStartStopCmdEnPa := emC_LUC[LUC_Num].SM.In.SchedulerStartStopCmdEnPa, LogDisPa := emC_LUC[LUC_Num].SM.In.LogDisPa, ClearLogEnPa := emC_LUC[LUC_Num].SM.In.ClearLogEnPa);
emC_LUC[LUC_Num].SM.Out.ManualMd := emC_E_StateMachine_1.ManualMd;
emC_LUC[LUC_Num].SM.Out.OperatorMd := emC_E_StateMachine_1.OperatorMd;
emC_LUC[LUC_Num].SM.Out.AutoMd := emC_E_StateMachine_1.AutoMd;
emC_LUC[LUC_Num].SM.Out.BatStartingSt := emC_E_StateMachine_1.BatStartingSt;
emC_LUC[LUC_Num].SM.Out.StartingSt := emC_E_StateMachine_1.StartingSt;
emC_LUC[LUC_Num].SM.Out.BatStoppingSt := emC_E_StateMachine_1.BatStoppingSt;
emC_LUC[LUC_Num].SM.Out.StoppingSt := emC_E_StateMachine_1.StoppingSt;
emC_LUC[LUC_Num].SM.Out.CoolingTimeActiveSt := emC_E_StateMachine_1.CoolingTimeActiveSt;
emC_LUC[LUC_Num].SM.Out.MinRunTImeActiveSt := emC_E_StateMachine_1.MinRunTimeActiveSt;
emC_LUC[LUC_Num].SM.Out.FailedToStartAl := emC_E_StateMachine_1.FailedToStartAl;
emC_LUC[LUC_Num].SM.Out.FailedToStopAl := emC_E_StateMachine_1.FailedToStopAl;
emC_LUC[LUC_Num].SM.Out.GcStartStopCmdOut := emC_E_StateMachine_1.GcStartStopCmdOut;
emC_LUC[LUC_Num].SM.Out.GcStartCmdOut := emC_E_StateMachine_1.GcStartCmdOut;
emC_LUC[LUC_Num].SM.Out.BatEnCmdOut := emC_E_StateMachine_1.BatEnCmdOut;
emC_LUC[LUC_Num].SM.Out.GcStopCmdOut := emC_E_StateMachine_1.GcStopCmdOut;
emC_LUC[LUC_Num].SM.Out.SchedulableSt := emC_E_StateMachine_1.SchedulableSt;
emC_LUC[LUC_Num].SM.Out.BatDisCmdOut := emC_E_StateMachine_1.BatDisCmdOut;
emC_LUC[LUC_Num].SM.Out.UnPSStartStopAlarm := emC_E_StateMachine_1.UnPSStartStopAlarm;
emC_LUC[LUC_Num].SM.Out.BatEnDisCmdOut := emC_E_StateMachine_1.BatEnDisCmdOut;
emC_LUC[LUC_Num].SM.Out.ExtInt := emC_E_StateMachine_1.ExtInt;
emC_LUC[LUC_Num].SM.Out.SMLog := emC_E_StateMachine_1.SMLog;
END_PROGRAM

PROGRAM emC_LUC_R03_CtrlLogic
  VAR
    LUC_BESS_Parameters_1 : emC_LUC_BESS_Parameters;
  END_VAR
  VAR_EXTERNAL
    emC_LUC : emC_LUC_Array;
    PLCMODE_RUN : BOOL;
  END_VAR
  VAR
    TON_5 : TON;
  END_VAR
  VAR_EXTERNAL
    LUC_Num : INT;
  END_VAR
  VAR
    LUC_BESS_Logic_1 : emC_LUC_BESS_Logic;
    emC_LUC_BESS_Logic_1 : emC_LUC_BESS_Logic;
    emC_LUC_BESS_Parameters_1 : emC_LUC_BESS_Parameters;
  END_VAR

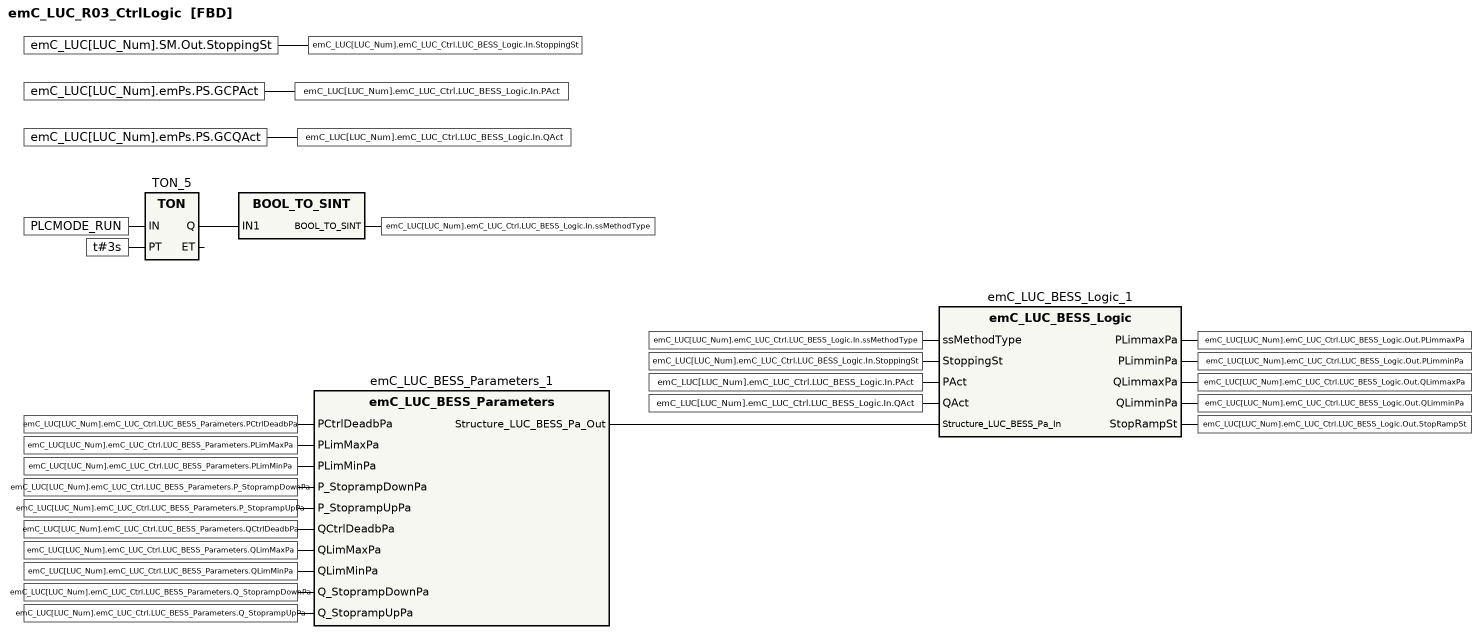
(* FBD diagram, written out as Structured Text *)
TON_5(IN := PLCMODE_RUN, PT := t#3s);
emC_LUC[LUC_Num].emC_LUC_Ctrl.LUC_BESS_Logic.In.ssMethodType := BOOL_TO_SINT(TON_5.Q);
emC_LUC[LUC_Num].emC_LUC_Ctrl.LUC_BESS_Logic.In.StoppingSt := emC_LUC[LUC_Num].SM.Out.StoppingSt;
emC_LUC[LUC_Num].emC_LUC_Ctrl.LUC_BESS_Logic.In.PAct := emC_LUC[LUC_Num].emPs.PS.GCPAct;
emC_LUC[LUC_Num].emC_LUC_Ctrl.LUC_BESS_Logic.In.QAct := emC_LUC[LUC_Num].emPs.PS.GCQAct;
emC_LUC_BESS_Parameters_1(PCtrlDeadbPa := emC_LUC[LUC_Num].emC_LUC_Ctrl.LUC_BESS_Parameters.PCtrlDeadbPa, PLimMaxPa := emC_LUC[LUC_Num].emC_LUC_Ctrl.LUC_BESS_Parameters.PLimMaxPa, PLimMinPa := emC_LUC[LUC_Num].emC_LUC_Ctrl.LUC_BESS_Parameters.PLimMinPa, P_StoprampDownPa := emC_LUC[LUC_Num].emC_LUC_Ctrl.LUC_BESS_Parameters.P_StoprampDownPa, P_StoprampUpPa := emC_LUC[LUC_Num].emC_LUC_Ctrl.LUC_BESS_Parameters.P_StoprampUpPa, QCtrlDeadbPa := emC_LUC[LUC_Num].emC_LUC_Ctrl.LUC_BESS_Parameters.QCtrlDeadbPa, QLimMaxPa := emC_LUC[LUC_Num].emC_LUC_Ctrl.LUC_BESS_Parameters.QLimMaxPa, QLimMinPa := emC_LUC[LUC_Num].emC_LUC_Ctrl.LUC_BESS_Parameters.QLimMinPa, Q_StoprampDownPa := emC_LUC[LUC_Num].emC_LUC_Ctrl.LUC_BESS_Parameters.Q_StoprampDownPa, Q_StoprampUpPa := emC_LUC[LUC_Num].emC_LUC_Ctrl.LUC_BESS_Parameters.Q_StoprampUpPa);
emC_LUC_BESS_Logic_1(ssMethodType := emC_LUC[LUC_Num].emC_LUC_Ctrl.LUC_BESS_Logic.In.ssMethodType, StoppingSt := emC_LUC[LUC_Num].emC_LUC_Ctrl.LUC_BESS_Logic.In.StoppingSt, PAct := emC_LUC[LUC_Num].emC_LUC_Ctrl.LUC_BESS_Logic.In.PAct, QAct := emC_LUC[LUC_Num].emC_LUC_Ctrl.LUC_BESS_Logic.In.QAct, Structure_LUC_BESS_Pa_In := emC_LUC_BESS_Parameters_1.Structure_LUC_BESS_Pa_Out);
emC_LUC[LUC_Num].emC_LUC_Ctrl.LUC_BESS_Logic.Out.PLimmaxPa := emC_LUC_BESS_Logic_1.PLimmaxPa;
emC_LUC[LUC_Num].emC_LUC_Ctrl.LUC_BESS_Logic.Out.PLimminPa := emC_LUC_BESS_Logic_1.PLimminPa;
emC_LUC[LUC_Num].emC_LUC_Ctrl.LUC_BESS_Logic.Out.QLimmaxPa := emC_LUC_BESS_Logic_1.QLimmaxPa;
emC_LUC[LUC_Num].emC_LUC_Ctrl.LUC_BESS_Logic.Out.QLimminPa := emC_LUC_BESS_Logic_1.QLimminPa;
emC_LUC[LUC_Num].emC_LUC_Ctrl.LUC_BESS_Logic.Out.StopRampSt := emC_LUC_BESS_Logic_1.StopRampSt;
END_PROGRAM

PROGRAM emC_LUC_R04_DevOut
  VAR
    emPS_Out_1 : emPS_Out;
    PSR_W_CMD_Q : TDC;
    PSR_W_CMD_I : TDC;
    PSR2_R_CMD_I : TDC;
    PSR2_R_CMD_Q : TDC;
    TON_5 : TON;
  END_VAR
  VAR_EXTERNAL
    LUC_Num : INT;
    emC_LUC : emC_LUC_Array;
    PLCMODE_RUN : BOOL;
  END_VAR
  VAR
    TestPset : REAL;
  END_VAR

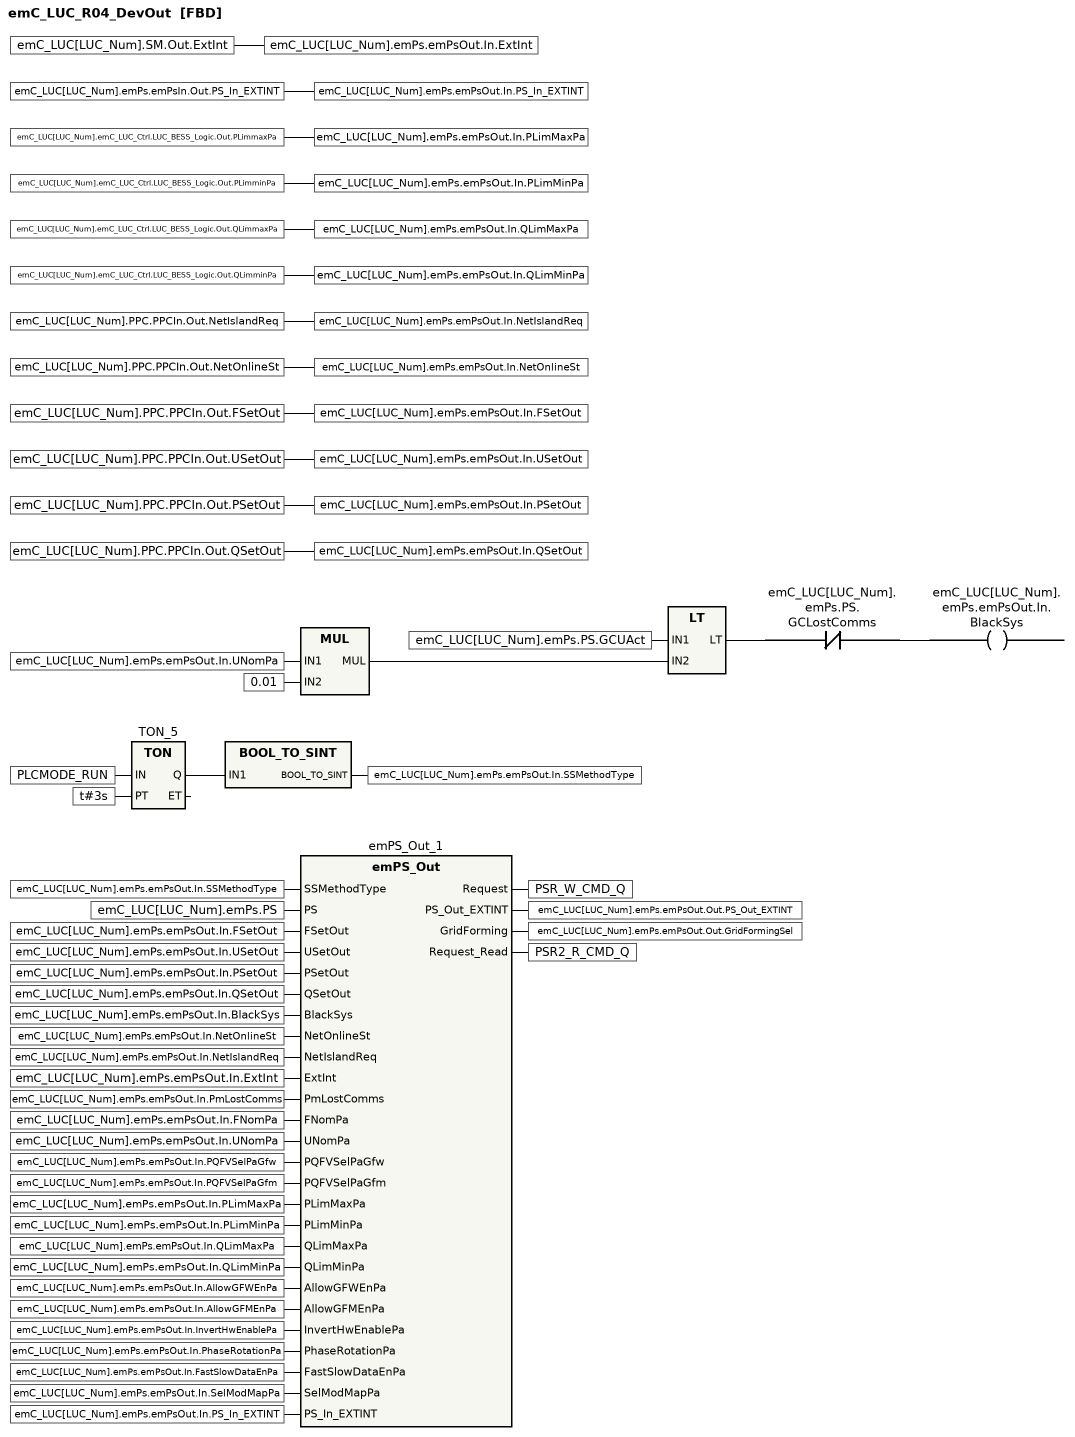
(* FBD diagram, written out as Structured Text *)
TON_5(IN := PLCMODE_RUN, PT := t#3s);
emC_LUC[LUC_Num].emPs.emPsOut.In.SSMethodType := BOOL_TO_SINT(TON_5.Q);
emC_LUC[LUC_Num].emPs.emPsOut.In.ExtInt := emC_LUC[LUC_Num].SM.Out.ExtInt;
emC_LUC[LUC_Num].emPs.emPsOut.In.PS_In_EXTINT := emC_LUC[LUC_Num].emPs.emPsIn.Out.PS_In_EXTINT;
emC_LUC[LUC_Num].emPs.emPsOut.In.BlackSys := emC_LUC[LUC_Num].emPs.PS.GCUAct < emC_LUC[LUC_Num].emPs.emPsOut.In.UNomPa * 0.01 AND NOT emC_LUC[LUC_Num].emPs.PS.GCLostComms;
emC_LUC[LUC_Num].emPs.emPsOut.In.PLimMinPa := emC_LUC[LUC_Num].emC_LUC_Ctrl.LUC_BESS_Logic.Out.PLimminPa;
emC_LUC[LUC_Num].emPs.emPsOut.In.PLimMaxPa := emC_LUC[LUC_Num].emC_LUC_Ctrl.LUC_BESS_Logic.Out.PLimmaxPa;
emC_LUC[LUC_Num].emPs.emPsOut.In.QLimMinPa := emC_LUC[LUC_Num].emC_LUC_Ctrl.LUC_BESS_Logic.Out.QLimminPa;
emC_LUC[LUC_Num].emPs.emPsOut.In.NetOnlineSt := emC_LUC[LUC_Num].PPC.PPCIn.Out.NetOnlineSt;
emC_LUC[LUC_Num].emPs.emPsOut.In.QLimMaxPa := emC_LUC[LUC_Num].emC_LUC_Ctrl.LUC_BESS_Logic.Out.QLimmaxPa;
emC_LUC[LUC_Num].emPs.emPsOut.In.NetIslandReq := emC_LUC[LUC_Num].PPC.PPCIn.Out.NetIslandReq;
emC_LUC[LUC_Num].emPs.emPsOut.In.USetOut := emC_LUC[LUC_Num].PPC.PPCIn.Out.USetOut;
emC_LUC[LUC_Num].emPs.emPsOut.In.PSetOut := emC_LUC[LUC_Num].PPC.PPCIn.Out.PSetOut;
emC_LUC[LUC_Num].emPs.emPsOut.In.FSetOut := emC_LUC[LUC_Num].PPC.PPCIn.Out.FSetOut;
emC_LUC[LUC_Num].emPs.emPsOut.In.QSetOut := emC_LUC[LUC_Num].PPC.PPCIn.Out.QSetOut;
emPS_Out_1(SSMethodType := emC_LUC[LUC_Num].emPs.emPsOut.In.SSMethodType, PS := emC_LUC[LUC_Num].emPs.PS, FSetOut := emC_LUC[LUC_Num].emPs.emPsOut.In.FSetOut, USetOut := emC_LUC[LUC_Num].emPs.emPsOut.In.USetOut, PSetOut := emC_LUC[LUC_Num].emPs.emPsOut.In.PSetOut, QSetOut := emC_LUC[LUC_Num].emPs.emPsOut.In.QSetOut, BlackSys := emC_LUC[LUC_Num].emPs.emPsOut.In.BlackSys, NetOnlineSt := emC_LUC[LUC_Num].emPs.emPsOut.In.NetOnlineSt, NetIslandReq := emC_LUC[LUC_Num].emPs.emPsOut.In.NetIslandReq, ExtInt := emC_LUC[LUC_Num].emPs.emPsOut.In.ExtInt, PmLostComms := emC_LUC[LUC_Num].emPs.emPsOut.In.PmLostComms, FNomPa := emC_LUC[LUC_Num].emPs.emPsOut.In.FNomPa, UNomPa := emC_LUC[LUC_Num].emPs.emPsOut.In.UNomPa, PQFVSelPaGfw := emC_LUC[LUC_Num].emPs.emPsOut.In.PQFVSelPaGfw, PQFVSelPaGfm := emC_LUC[LUC_Num].emPs.emPsOut.In.PQFVSelPaGfm, PLimMaxPa := emC_LUC[LUC_Num].emPs.emPsOut.In.PLimMaxPa, PLimMinPa := emC_LUC[LUC_Num].emPs.emPsOut.In.PLimMinPa, QLimMaxPa := emC_LUC[LUC_Num].emPs.emPsOut.In.QLimMaxPa, QLimMinPa := emC_LUC[LUC_Num].emPs.emPsOut.In.QLimMinPa, AllowGFWEnPa := emC_LUC[LUC_Num].emPs.emPsOut.In.AllowGFWEnPa, AllowGFMEnPa := emC_LUC[LUC_Num].emPs.emPsOut.In.AllowGFMEnPa, InvertHwEnablePa := emC_LUC[LUC_Num].emPs.emPsOut.In.InvertHwEnablePa, PhaseRotationPa := emC_LUC[LUC_Num].emPs.emPsOut.In.PhaseRotationPa, FastSlowDataEnPa := emC_LUC[LUC_Num].emPs.emPsOut.In.FastSlowDataEnPa, SelModMapPa := emC_LUC[LUC_Num].emPs.emPsOut.In.SelModMapPa, PS_In_EXTINT := emC_LUC[LUC_Num].emPs.emPsOut.In.PS_In_EXTINT);
PSR_W_CMD_Q := emPS_Out_1.Request;
PSR2_R_CMD_Q := emPS_Out_1.Request_Read;
emC_LUC[LUC_Num].emPs.emPsOut.Out.PS_Out_EXTINT := emPS_Out_1.PS_Out_EXTINT;
emC_LUC[LUC_Num].emPs.emPsOut.Out.GridFormingSel := emPS_Out_1.GridForming;
END_PROGRAM

PROGRAM emC_LUC_R05_MSH_Out
  VAR
    S_SPI_MNG_1001 : S_SPI_MNG;
    S_SPI_MNG_1002 : S_SPI_MNG;
    S_SPI_MNG_1003 : S_SPI_MNG;
    S_SPI_MNG_1004 : S_SPI_MNG;
    S_SPI_MNG_1005 : S_SPI_MNG;
    S_SPI_MNG_1006 : S_SPI_MNG;
    S_SPI_MNG_1007 : S_SPI_MNG;
    PPC_GCFaultSt_Q : SPI;
    PPC_NonCriticalAl_Q : SPI;
    PPC_CriticalAl_Q : SPI;
    PPC_WarningAl_Q : SPI;
    PPC_StoppingSt_Q : SPI;
    PPC_CtrlSystemReady_Q : SPI;
    PPC_BlackSys_Q : SPI;
    S_MFI_MNG_1001 : S_MFI_MNG;
    S_MFI_MNG_1002 : S_MFI_MNG;
    S_MFI_MNG_1003 : S_MFI_MNG;
    S_MFI_MNG_1004 : S_MFI_MNG;
    S_MFI_MNG_1005 : S_MFI_MNG;
    S_MFI_MNG_1006 : S_MFI_MNG;
    S_MFI_MNG_1007 : S_MFI_MNG;
    S_MFI_MNG_1008 : S_MFI_MNG;
    PPC_TempAct_Q : MFI;
    PPC_BatPNomMaxAct_Q : MFI;
    PPC_BatPNomMinAct_Q : MFI;
    PPC_BatSocAct_Q : MFI;
    PPC_UAct_Q : MFI;
    PPC_FAct_Q : MFI;
    PPC_PAct_Q : MFI;
    PPC_QAct_Q : MFI;
    S_SPI_MNG_1008 : S_SPI_MNG;
    S_SPI_MNG_1009 : S_SPI_MNG;
    PPC_OnlineSt_Q : SPI;
    PPC_RunningSt_Q : SPI;
    i : INT;
    GCI1_Q : MFI;
    GCI2_Q : MFI;
    GCI3_Q : MFI;
    S_MFI_MNG_64 : S_MFI_MNG;
    S_MFI_MNG_63 : S_MFI_MNG;
    TimeStamp : Timestamp;
    S_SPI_MNG_1 : S_SPI_MNG;
    S_SPI_MNG_2 : S_SPI_MNG;
    S_SPI_MNG_3 : S_SPI_MNG;
    S_SPI_MNG_5 : S_SPI_MNG;
    S_SPI_MNG_6 : S_SPI_MNG;
    S_SPI_MNG_7 : S_SPI_MNG;
    S_SPI_MNG_8 : S_SPI_MNG;
    S_SPI_MNG_9 : S_SPI_MNG;
    S_SPI_MNG_10 : S_SPI_MNG;
    S_SPI_MNG_14 : S_SPI_MNG;
    S_SPI_MNG_19 : S_SPI_MNG;
    S_SPI_MNG_20 : S_SPI_MNG;
    S_SPI_MNG_21 : S_SPI_MNG;
    S_SPI_MNG_22 : S_SPI_MNG;
    S_SPI_MNG_23 : S_SPI_MNG;
    S_SPI_MNG_24 : S_SPI_MNG;
    S_SPI_MNG_25 : S_SPI_MNG;
    S_SPI_MNG_26 : S_SPI_MNG;
    S_SPI_MNG_27 : S_SPI_MNG;
    S_SPI_MNG_28 : S_SPI_MNG;
    S_SPI_MNG_29 : S_SPI_MNG;
    S_SPI_MNG_30 : S_SPI_MNG;
    S_SPI_MNG_31 : S_SPI_MNG;
    S_SPI_MNG_32 : S_SPI_MNG;
    S_SPI_MNG_33 : S_SPI_MNG;
    S_SPI_MNG_34 : S_SPI_MNG;
    S_SPI_MNG_35 : S_SPI_MNG;
    S_SPI_MNG_36 : S_SPI_MNG;
    S_SPI_MNG_37 : S_SPI_MNG;
    S_SPI_MNG_38 : S_SPI_MNG;
    S_SPI_MNG_39 : S_SPI_MNG;
    S_SPI_MNG_40 : S_SPI_MNG;
    S_SPI_MNG_41 : S_SPI_MNG;
    S_SPI_MNG_42 : S_SPI_MNG;
    S_SPI_MNG_43 : S_SPI_MNG;
    S_SPI_MNG_44 : S_SPI_MNG;
    S_SPI_MNG_45 : S_SPI_MNG;
    S_SPI_MNG_46 : S_SPI_MNG;
    S_SPI_MNG_47 : S_SPI_MNG;
    S_SPI_MNG_48 : S_SPI_MNG;
    S_SPI_MNG_49 : S_SPI_MNG;
    S_SPI_MNG_50 : S_SPI_MNG;
    S_SPI_MNG_51 : S_SPI_MNG;
    S_SPI_MNG_52 : S_SPI_MNG;
    S_SPI_MNG_53 : S_SPI_MNG;
    S_SPI_MNG_54 : S_SPI_MNG;
    S_SPI_MNG_55 : S_SPI_MNG;
    S_SPI_MNG_56 : S_SPI_MNG;
    S_SPI_MNG_57 : S_SPI_MNG;
    S_SPI_MNG_58 : S_SPI_MNG;
    S_SPI_MNG_59 : S_SPI_MNG;
    S_SPI_MNG_60 : S_SPI_MNG;
    S_SPI_MNG_61 : S_SPI_MNG;
    S_SPI_MNG_62 : S_SPI_MNG;
    S_SPI_MNG_63 : S_SPI_MNG;
    S_SPI_MNG_64 : S_SPI_MNG;
    S_SPI_MNG_65 : S_SPI_MNG;
    S_SPI_MNG_66 : S_SPI_MNG;
    S_SPI_MNG_67 : S_SPI_MNG;
    S_SPI_MNG_68 : S_SPI_MNG;
    S_SPI_MNG_69 : S_SPI_MNG;
    S_SPI_MNG_70 : S_SPI_MNG;
    S_SPI_MNG_71 : S_SPI_MNG;
    S_SPI_MNG_72 : S_SPI_MNG;
    S_SPI_MNG_73 : S_SPI_MNG;
    S_SPI_MNG_74 : S_SPI_MNG;
    S_SPI_MNG_75 : S_SPI_MNG;
    S_SPI_MNG_76 : S_SPI_MNG;
    S_SPI_MNG_77 : S_SPI_MNG;
    S_SPI_MNG_78 : S_SPI_MNG;
    S_SPI_MNG_79 : S_SPI_MNG;
    S_SPI_MNG_80 : S_SPI_MNG;
    S_SPI_MNG_81 : S_SPI_MNG;
    S_SPI_MNG_82 : S_SPI_MNG;
    S_SPI_MNG_83 : S_SPI_MNG;
    S_SPI_MNG_84 : S_SPI_MNG;
    S_SPI_MNG_85 : S_SPI_MNG;
    S_SPI_MNG_86 : S_SPI_MNG;
    S_SPI_MNG_87 : S_SPI_MNG;
    S_SPI_MNG_88 : S_SPI_MNG;
    S_SPI_MNG_89 : S_SPI_MNG;
    S_SPI_MNG_90 : S_SPI_MNG;
    S_SPI_MNG_91 : S_SPI_MNG;
    S_SPI_MNG_92 : S_SPI_MNG;
    S_SPI_MNG_93 : S_SPI_MNG;
    S_SPI_MNG_94 : S_SPI_MNG;
    S_SPI_MNG_95 : S_SPI_MNG;
    S_SPI_MNG_96 : S_SPI_MNG;
    S_SPI_MNG_97 : S_SPI_MNG;
    S_SPI_MNG_98 : S_SPI_MNG;
    S_SPI_MNG_99 : S_SPI_MNG;
    S_SPI_MNG_100 : S_SPI_MNG;
    S_SPI_MNG_101 : S_SPI_MNG;
    S_SPI_MNG_102 : S_SPI_MNG;
    S_SPI_MNG_103 : S_SPI_MNG;
    S_SPI_MNG_104 : S_SPI_MNG;
    S_SPI_MNG_105 : S_SPI_MNG;
    S_SPI_MNG_106 : S_SPI_MNG;
    S_SPI_MNG_107 : S_SPI_MNG;
    S_SPI_MNG_108 : S_SPI_MNG;
    S_SPI_MNG_109 : S_SPI_MNG;
    S_SPI_MNG_110 : S_SPI_MNG;
    S_SPI_MNG_111 : S_SPI_MNG;
    S_SPI_MNG_112 : S_SPI_MNG;
    S_SPI_MNG_113 : S_SPI_MNG;
    S_SPI_MNG_114 : S_SPI_MNG;
    S_SPI_MNG_115 : S_SPI_MNG;
    S_SPI_MNG_116 : S_SPI_MNG;
    RTU_RTC_1 : RTU_RTC;
  END_VAR
  VAR_EXTERNAL
    emC_LUC : emC_LUC_Array;
    LUC_Num : INT;
  END_VAR
  VAR
    OperatorMd_Q : SPI;
    AutoMd_Q : SPI;
    LocalOnlineSt_Q : SPI;
    StoppedSt_Q : SPI;
    ManualMd_Q : SPI;
    FailedToStartAl_Q : SPI;
    FailedToStopAl_Q : SPI;
    NonCriticalAl_Q : SPI;
    WarningAl_Q : SPI;
    CriticalAl_Q : SPI;
    AcCbOpenAl_Q : SPI;
    AcCbCloseAl_Q : SPI;
    AcCbClosedSt_Q : SPI;
    EstopAl_Q : SPI;
    InsulAl_Q : SPI;
    AuxSplyLossAl_Q : SPI;
    GcDcEqAl_Q : SPI;
    GcCriticalAl_Q : SPI;
    FaultAl_Q : SPI;
    HealthySt_Q : SPI;
    OnlineSt_Q : SPI;
    RunningSt_Q : SPI;
    BatEmergencyStop_Q : SPI;
    BlackOutCondition_Q : SPI;
    BatInitializeSt_Q : SPI;
    BatNotReadySt_Q : SPI;
    BatReadySt_Q : SPI;
    BatStartingSt_Q : SPI;
    BatOnlineSt_Q : SPI;
    BatStoppingSt_Q : SPI;
    BmsEStopProtEn_Q : SPI;
    BmsEStopSPDEn_Q : SPI;
    BmsChargingSt_Q : SPI;
    BmsDischargingSt_Q : SPI;
    BattRunningSt_Q : SPI;
    BmsRkPartOnlineSt_Q : SPI;
    BmsEStopSPDSt_Q : SPI;
    BmsEStopProtSt_Q : SPI;
    BmsEStopPartSt_Q : SPI;
    BmsHealthySt_Q : SPI;
    BmsFireSysOkSt_Q : SPI;
    BmsCriticalAl_Q : SPI;
    BmsNonCriticalAl_Q : SPI;
    BmsWarningAl_Q : SPI;
    BmsStateTOUT_Q : SPI;
    BmsInitCommsFail_Q : SPI;
    BmsMinRkCloseFail_Q : SPI;
    BmsRkTripStart_Q : SPI;
    BmsMinRkOnlineFail_Q : SPI;
    BmsRkFailToOpen_Q : SPI;
    BmsSysFireAl_Q : SPI;
    BmsBmsLostCommsAl_Q : SPI;
    BmsBankFault_Q : SPI;
    BmsEStopAl_Q : SPI;
    BmsExtReadyStNotSetAl_Q : SPI;
    BattUSyncErrAl_Q : SPI;
    BmsRkFail2Cls_Q : SPI;
    BmsRkCntrFailAl_Q : SPI;
    BmsRTUComAl_Q : SPI;
    BmsRTUComFlt_Q : SPI;
    BmsRkVoltImbAl_Q : SPI;
    BmsSysStopAl_Q : SPI;
    BmsModuleUnderTempAl_Q : SPI;
    BmsModuleOverTempAl_Q : SPI;
    BmsModuleUnVoltAl_Q : SPI;
    BmsModuleOvVoltAl_Q : SPI;
    BmsRackVoltRegAl_Q : SPI;
    BmsRackTempRegAl_Q : SPI;
    BmsAuxProtAl_Q : SPI;
    BmsChargeOperLimAl_Q : SPI;
    BmsDischargeOperLimAl_Q : SPI;
    BmsRackUnVoltAl_Q : SPI;
    BmsRackOvVoltAl_Q : SPI;
    BmsRackCommsAl_Q : SPI;
    BmsTrayCommsAl_Q : SPI;
    BmsDcCntrSensor1Al_Q : SPI;
    BmsDcCntrSensor2Al_Q : SPI;
    BmsFanFailAl_Q : SPI;
    BmsChargeOverCurrentAl_Q : SPI;
    BmsDisChargeOverCurrentAl_Q : SPI;
    BmsRackVSenseDiffAl_Q : SPI;
    BmsRackFuseFailAl_Q : SPI;
    BmsRackCurrentSenserFailAl_Q : SPI;
    BmsRackPermanentUVAl_Q : SPI;
    BmsDcCntr1Al_Q : SPI;
    BmsDcCntr2Al_Q : SPI;
    BmsDcSwCntFailAl_Q : SPI;
    BmsCellVoltSenFailAl_Q : SPI;
    BmsDCFuseSenserFailAl_Q : SPI;
    BmsModuleUnderTempProt_Q : SPI;
    BmsModuleOverTempProt_Q : SPI;
    BmsModuleUnVoltProt_Q : SPI;
    BmsModuleOvVoltProt_Q : SPI;
    BmsRackVoltRegProt_Q : SPI;
    BmsRackTempRegProt_Q : SPI;
    BmsAuxProtProt_Q : SPI;
    BmsChargeOperLimProt_Q : SPI;
    BmsDischargeOperLimProt_Q : SPI;
    BmsRackUnVoltProt_Q : SPI;
    BmsRackOvVoltProt_Q : SPI;
    BmsRackCommsProt_Q : SPI;
    BmsTrayCommsProt_Q : SPI;
    BmsDcCntrSensor1Prot_Q : SPI;
    BmsDcCntrSensor2Prot_Q : SPI;
    BmsFanFailProt_Q : SPI;
    BmsChargeOverCurrentProt_Q : SPI;
    BmsDisChargeOverCurrentProt_Q : SPI;
    BmsRackVSenseDiffProt_Q : SPI;
    BmsRackFuseFailProt_Q : SPI;
    BmsRackCurrentSenserFailProt_Q : SPI;
    BmsRackPermanentUVProt_Q : SPI;
    BmsDcCntr1Prot_Q : SPI;
    BmsDcCntr2Prot_Q : SPI;
    BmsDcSwCntFailProt_Q : SPI;
    BmsCellVoltSenFailProt_Q : SPI;
    BmsDCFuseSenserFailProt_Q : SPI;
    U12Act_Q : MFI;
    U23Act_Q : MFI;
    U31Act_Q : MFI;
    I1Act_Q : MFI;
    I2Act_Q : MFI;
    I3Act_Q : MFI;
    PfAct_Q : MFI;
    TempAct_Q : MFI;
    UAct_Q : MFI;
    PAct_Q : MFI;
    QAct_Q : MFI;
    EAct_Q : MFI;
    FAct_Q : MFI;
    GcSPNomAct_Q : MFI;
    GcINomAct_Q : MFI;
    GcUNomAct_Q : MFI;
    GcFNomAct_Q : MFI;
    GcModUNomAct_Q : MFI;
    BatPNomMinAct_Q : MFI;
    BmsChrgMwhAct_Q : MFI;
    BmsServVolt_Q : MFI;
    S_SPI_MNG_117 : S_SPI_MNG;
    S_SPI_MNG_118 : S_SPI_MNG;
    S_SPI_MNG_119 : S_SPI_MNG;
    S_SPI_MNG_120 : S_SPI_MNG;
    S_SPI_MNG_121 : S_SPI_MNG;
    S_SPI_MNG_122 : S_SPI_MNG;
    S_SPI_MNG_123 : S_SPI_MNG;
    S_SPI_MNG_124 : S_SPI_MNG;
    S_SPI_MNG_125 : S_SPI_MNG;
    S_SPI_MNG_126 : S_SPI_MNG;
    S_SPI_MNG_127 : S_SPI_MNG;
    S_SPI_MNG_128 : S_SPI_MNG;
    S_SPI_MNG_129 : S_SPI_MNG;
    S_SPI_MNG_130 : S_SPI_MNG;
    S_SPI_MNG_131 : S_SPI_MNG;
    S_SPI_MNG_132 : S_SPI_MNG;
    S_SPI_MNG_133 : S_SPI_MNG;
    S_SPI_MNG_134 : S_SPI_MNG;
    S_SPI_MNG_135 : S_SPI_MNG;
    S_SPI_MNG_136 : S_SPI_MNG;
    S_SPI_MNG_137 : S_SPI_MNG;
    S_SPI_MNG_138 : S_SPI_MNG;
    S_SPI_MNG_139 : S_SPI_MNG;
    S_SPI_MNG_140 : S_SPI_MNG;
    S_SPI_MNG_141 : S_SPI_MNG;
    S_SPI_MNG_142 : S_SPI_MNG;
    S_SPI_MNG_143 : S_SPI_MNG;
    S_SPI_MNG_162 : S_SPI_MNG;
    S_SPI_MNG_163 : S_SPI_MNG;
    S_SPI_MNG_164 : S_SPI_MNG;
    S_SPI_MNG_165 : S_SPI_MNG;
    S_SPI_MNG_166 : S_SPI_MNG;
    S_SPI_MNG_167 : S_SPI_MNG;
    S_SPI_MNG_168 : S_SPI_MNG;
    S_SPI_MNG_169 : S_SPI_MNG;
    S_SPI_MNG_172 : S_SPI_MNG;
    S_SPI_MNG_173 : S_SPI_MNG;
    S_SPI_MNG_174 : S_SPI_MNG;
    S_SPI_MNG_175 : S_SPI_MNG;
    S_SPI_MNG_176 : S_SPI_MNG;
    S_SPI_MNG_177 : S_SPI_MNG;
    S_SPI_MNG_178 : S_SPI_MNG;
    S_SPI_MNG_179 : S_SPI_MNG;
    S_SPI_MNG_180 : S_SPI_MNG;
    S_SPI_MNG_181 : S_SPI_MNG;
    S_SPI_MNG_182 : S_SPI_MNG;
    S_SPI_MNG_183 : S_SPI_MNG;
    S_SPI_MNG_184 : S_SPI_MNG;
    S_SPI_MNG_185 : S_SPI_MNG;
    S_SPI_MNG_186 : S_SPI_MNG;
    S_SPI_MNG_187 : S_SPI_MNG;
    S_SPI_MNG_188 : S_SPI_MNG;
    S_SPI_MNG_189 : S_SPI_MNG;
    S_SPI_MNG_190 : S_SPI_MNG;
    S_SPI_MNG_191 : S_SPI_MNG;
    S_SPI_MNG_192 : S_SPI_MNG;
    S_SPI_MNG_193 : S_SPI_MNG;
    S_SPI_MNG_194 : S_SPI_MNG;
    S_SPI_MNG_195 : S_SPI_MNG;
    S_SPI_MNG_196 : S_SPI_MNG;
    S_SPI_MNG_197 : S_SPI_MNG;
    S_SPI_MNG_198 : S_SPI_MNG;
    S_SPI_MNG_199 : S_SPI_MNG;
    S_SPI_MNG_200 : S_SPI_MNG;
    S_SPI_MNG_201 : S_SPI_MNG;
    S_SPI_MNG_202 : S_SPI_MNG;
    S_SPI_MNG_203 : S_SPI_MNG;
    S_SPI_MNG_205 : S_SPI_MNG;
    S_SPI_MNG_206 : S_SPI_MNG;
    S_SPI_MNG_207 : S_SPI_MNG;
    S_SPI_MNG_208 : S_SPI_MNG;
    S_SPI_MNG_209 : S_SPI_MNG;
    S_SPI_MNG_210 : S_SPI_MNG;
    S_SPI_MNG_211 : S_SPI_MNG;
    S_SPI_MNG_212 : S_SPI_MNG;
    S_SPI_MNG_213 : S_SPI_MNG;
    S_SPI_MNG_214 : S_SPI_MNG;
    S_SPI_MNG_215 : S_SPI_MNG;
    S_SPI_MNG_216 : S_SPI_MNG;
    S_SPI_MNG_217 : S_SPI_MNG;
    S_SPI_MNG_218 : S_SPI_MNG;
    S_SPI_MNG_219 : S_SPI_MNG;
    S_SPI_MNG_220 : S_SPI_MNG;
    S_SPI_MNG_221 : S_SPI_MNG;
    S_SPI_MNG_222 : S_SPI_MNG;
    S_SPI_MNG_223 : S_SPI_MNG;
    S_SPI_MNG_224 : S_SPI_MNG;
    S_SPI_MNG_225 : S_SPI_MNG;
    S_SPI_MNG_226 : S_SPI_MNG;
    S_SPI_MNG_227 : S_SPI_MNG;
    S_SPI_MNG_228 : S_SPI_MNG;
    S_SPI_MNG_229 : S_SPI_MNG;
    S_SPI_MNG_230 : S_SPI_MNG;
    S_SPI_MNG_231 : S_SPI_MNG;
    S_SPI_MNG_232 : S_SPI_MNG;
    S_SPI_MNG_233 : S_SPI_MNG;
    S_SPI_MNG_234 : S_SPI_MNG;
    S_SPI_MNG_235 : S_SPI_MNG;
    S_SPI_MNG_236 : S_SPI_MNG;
    S_SPI_MNG_237 : S_SPI_MNG;
    S_SPI_MNG_238 : S_SPI_MNG;
    S_SPI_MNG_239 : S_SPI_MNG;
    S_SPI_MNG_240 : S_SPI_MNG;
    S_SPI_MNG_241 : S_SPI_MNG;
    S_SPI_MNG_242 : S_SPI_MNG;
    S_SPI_MNG_243 : S_SPI_MNG;
    S_SPI_MNG_244 : S_SPI_MNG;
    S_SPI_MNG_245 : S_SPI_MNG;
    S_SPI_MNG_246 : S_SPI_MNG;
    S_SPI_MNG_247 : S_SPI_MNG;
    S_SPI_MNG_248 : S_SPI_MNG;
    S_SPI_MNG_249 : S_SPI_MNG;
    S_SPI_MNG_250 : S_SPI_MNG;
    S_SPI_MNG_251 : S_SPI_MNG;
    S_SPI_MNG_252 : S_SPI_MNG;
    S_SPI_MNG_253 : S_SPI_MNG;
    S_SPI_MNG_254 : S_SPI_MNG;
    S_SPI_MNG_255 : S_SPI_MNG;
    S_SPI_MNG_256 : S_SPI_MNG;
    S_SPI_MNG_257 : S_SPI_MNG;
    S_SPI_MNG_258 : S_SPI_MNG;
    S_SPI_MNG_259 : S_SPI_MNG;
    S_SPI_MNG_260 : S_SPI_MNG;
    S_SPI_MNG_261 : S_SPI_MNG;
    S_SPI_MNG_262 : S_SPI_MNG;
    S_SPI_MNG_263 : S_SPI_MNG;
    S_SPI_MNG_264 : S_SPI_MNG;
    S_SPI_MNG_265 : S_SPI_MNG;
    S_SPI_MNG_266 : S_SPI_MNG;
    S_SPI_MNG_267 : S_SPI_MNG;
    S_SPI_MNG_268 : S_SPI_MNG;
    S_SPI_MNG_269 : S_SPI_MNG;
    S_SPI_MNG_270 : S_SPI_MNG;
    S_SPI_MNG_271 : S_SPI_MNG;
    S_SPI_MNG_272 : S_SPI_MNG;
    S_SPI_MNG_273 : S_SPI_MNG;
    GCRunningSt_Q : SPI;
    GCHealthy_Q : SPI;
    GCStartingSt_Q : SPI;
    GCReadySt_Q : SPI;
    GCGridFollowing_Q : SPI;
    GCFaultSt_Q : SPI;
    GCGridForming_Q : SPI;
    GCAreaEPSLost_Q : SPI;
    GCChargingSt_Q : SPI;
    GCRideThru_Q : SPI;
    GCTransitionActiveSt_Q : SPI;
    GCGndFault_Q : SPI;
    GCDCOverU_Q : SPI;
    GCACDisconnect_Q : SPI;
    GCDCDisconnect_Q : SPI;
    GCDCGridDisconnect_Q : SPI;
    GCCabinetOpen_Q : SPI;
    GCManualShutdown_Q : SPI;
    GCOverTemp_Q : SPI;
    GCOverF_Q : SPI;
    GCUnderF_Q : SPI;
    GCACOverVolt_Q : SPI;
    GCACUnderVolt_Q : SPI;
    GCBlownFuse_Q : SPI;
    GCUnderTemp_Q : SPI;
    GCMemLoss_Q : SPI;
    GCHWTestFailed_Q : SPI;
    GCABBCtrlWrongConfig_Q : SPI;
    GCABBCtrlReady_Q : SPI;
    GCABBCtrlStartingSt_Q : SPI;
    GCABBCtrlVGMActiveSt_Q : SPI;
    GCABBCtrlGSMActiveSt_Q : SPI;
    GCABBCtrlError_Q : SPI;
    GCABBCtrlStoppingSt_Q : SPI;
    GCABBCtrlIslanded_Q : SPI;
    GCLostComms_Q : SPI;
    GCCommsOk_Q : SPI;
    GCHardwareenablestatus_Q : SPI;
    GCACPowerAvailable_Q : SPI;
    GCDCPowerAvailable_Q : SPI;
    GCPowerCircuitEnabled_Q : SPI;
    GCMX1relaystatus_Q : SPI;
    GCMX2relaystatus_Q : SPI;
    GCPrechargestatus_Q : SPI;
    GCK2Relaystatus_Q : SPI;
    GCControlcommandsvalid_Q : SPI;
    GCPowercommandValid_Q : SPI;
    GCCurrentcommandValid_Q : SPI;
    GCPhaserotationstatus_Q : SPI;
    GCLinevoltagedetected_Q : SPI;
    GCUnused_Q : SPI;
    GCRemoteACPowerAvailable_Q : SPI;
    GCRemotephaserotationstatus_Q : SPI;
    GCRemoteLineVoltageDetected_Q : SPI;
    GCDI1Status_Q : SPI;
    GCDI2Status_Q : SPI;
    GCDI3Status_Q : SPI;
    GCDI4Status_Q : SPI;
    GCDO1Status_Q : SPI;
    GCDO2Status_Q : SPI;
    GCDO3Status_Q : SPI;
    GCDO4Status_Q : SPI;
    GCDClinkRefCmdValid_Q : SPI;
    GCPumpRunning_Q : SPI;
    GCPumpFault_Q : SPI;
    GCABBLostCommsStop_Q : SPI;
    CtrlSystemReady_Q : SPI;
    GCFlt_Estp_Q : SPI;
    GCFlt_ACOverCurrent_Q : SPI;
    GCFlt_DCOverCurrent_Q : SPI;
    GCFlt_DCOverVoltage_Q : SPI;
    GCFlt_PDOverTemp_Q : SPI;
    GCFlt_InvOverTemp_Q : SPI;
    GCFlt_CmdMsg_Q : SPI;
    GCFlt_DCUnderVolt_Q : SPI;
    GCFlt_ACOverVolt_Q : SPI;
    GCFlt_IllegalTrans_Q : SPI;
    GCFlt_EEHeat_Q : SPI;
    GCFlt_EESction_Q : SPI;
    GCFlt_Cool_Q : SPI;
    GCFlt_TimedOverLoadAC_Q : SPI;
    GCFlt_TimedOverLoadDC_Q : SPI;
    GCFlt_ICOL_Q : SPI;
    GCFlt_CtlBdVolt_Q : SPI;
    GCFlt_PChImbal_Q : SPI;
    GCFlt_DiDt_Q : SPI;
    GCFlt_CoolingFlw_Q : SPI;
    GCFlt_ThrmOverLoad_Q : SPI;
    GCFlt_Fan_Q : SPI;
    GCFlt_POR_Q : SPI;
    GCFlt_Condensation_Q : SPI;
    GCFlt_I2C_Q : SPI;
    GCFlt_ExternalInhibit_Q : SPI;
    GCFlt_GroundFault_Q : SPI;
    GCFlt_Fuse_Q : SPI;
    GCFlt_Rsvd28_Q : SPI;
    GCFlt_ACDisconnect_Q : SPI;
    GCFlt_Rsvd30_Q : SPI;
    GCFlt_Rsvd31_Q : SPI;
    GCWrn_CANW_Q : SPI;
    GCWrn_CANEP_Q : SPI;
    GCWrn_Thrm_Q : SPI;
    GCWrn_Fan_Q : SPI;
    GCWrn_EeSaveActive_Q : SPI;
    GCWrn_LocNetMismatch_Q : SPI;
    GCWrn_RemNetMismatch_Q : SPI;
    GCWrn_Condensation_Q : SPI;
    GCWrn_I2C_Q : SPI;
    GCWrn_ExternalInhibit_Q : SPI;
    GCWrn_MaintReqd_Q : SPI;
    GCWrn_GroundFault_Q : SPI;
    GCWrn_Fuse_Q : SPI;
    GCWrn_ACDisconnect_Q : SPI;
    GCWrn_Rsvd14_Q : SPI;
    GCWrn_Rsvd15_Q : SPI;
    GCWrn_Rsvd16_Q : SPI;
    GCWrn_Rsvd17_Q : SPI;
    GCWrn_Rsvd18_Q : SPI;
    GCWrn_Rsvd19_Q : SPI;
    GCWrn_Rsvd20_Q : SPI;
    GCWrn_Rsvd21_Q : SPI;
    GCWrn_Rsvd22_Q : SPI;
    GCWrn_Rsvd23_Q : SPI;
    GCWrn_Rsvd24_Q : SPI;
    GCWrn_Rsvd25_Q : SPI;
    GCWrn_Rsvd26_Q : SPI;
    GCWrn_Rsvd27_Q : SPI;
    GCWrn_Rsvd28_Q : SPI;
    GCWrn_Rsvd29_Q : SPI;
    GCWrn_Rsvd30_Q : SPI;
    GCCriticalAlarm_Q : SPI;
    GCNonCriticalAlarm_Q : SPI;
    GCWarning_Q : SPI;
    GCreconnectDelay_Q : SPI;
    GCMomentCessation_Q : SPI;
    GCInhibited_Q : SPI;
    S_MFI_MNG_1 : S_MFI_MNG;
    S_MFI_MNG_2 : S_MFI_MNG;
    S_MFI_MNG_3 : S_MFI_MNG;
    S_MFI_MNG_4 : S_MFI_MNG;
    S_MFI_MNG_5 : S_MFI_MNG;
    S_MFI_MNG_6 : S_MFI_MNG;
    S_MFI_MNG_7 : S_MFI_MNG;
    S_MFI_MNG_8 : S_MFI_MNG;
    S_MFI_MNG_9 : S_MFI_MNG;
    S_MFI_MNG_10 : S_MFI_MNG;
    S_MFI_MNG_11 : S_MFI_MNG;
    S_MFI_MNG_12 : S_MFI_MNG;
    S_MFI_MNG_13 : S_MFI_MNG;
    S_MFI_MNG_14 : S_MFI_MNG;
    S_MFI_MNG_15 : S_MFI_MNG;
    S_MFI_MNG_16 : S_MFI_MNG;
    S_MFI_MNG_17 : S_MFI_MNG;
    S_MFI_MNG_18 : S_MFI_MNG;
    S_MFI_MNG_19 : S_MFI_MNG;
    S_MFI_MNG_20 : S_MFI_MNG;
    S_MFI_MNG_21 : S_MFI_MNG;
    S_MFI_MNG_22 : S_MFI_MNG;
    S_MFI_MNG_23 : S_MFI_MNG;
    S_MFI_MNG_24 : S_MFI_MNG;
    S_MFI_MNG_25 : S_MFI_MNG;
    S_MFI_MNG_26 : S_MFI_MNG;
    S_MFI_MNG_27 : S_MFI_MNG;
    S_MFI_MNG_28 : S_MFI_MNG;
    S_MFI_MNG_29 : S_MFI_MNG;
    S_MFI_MNG_30 : S_MFI_MNG;
    S_MFI_MNG_31 : S_MFI_MNG;
    S_MFI_MNG_32 : S_MFI_MNG;
    S_MFI_MNG_33 : S_MFI_MNG;
    S_MFI_MNG_34 : S_MFI_MNG;
    S_MFI_MNG_35 : S_MFI_MNG;
    S_MFI_MNG_36 : S_MFI_MNG;
    S_MFI_MNG_37 : S_MFI_MNG;
    S_MFI_MNG_38 : S_MFI_MNG;
    S_MFI_MNG_39 : S_MFI_MNG;
    S_MFI_MNG_40 : S_MFI_MNG;
    S_MFI_MNG_41 : S_MFI_MNG;
    S_MFI_MNG_42 : S_MFI_MNG;
    S_MFI_MNG_43 : S_MFI_MNG;
    S_MFI_MNG_44 : S_MFI_MNG;
    S_MFI_MNG_45 : S_MFI_MNG;
    S_MFI_MNG_46 : S_MFI_MNG;
    S_MFI_MNG_47 : S_MFI_MNG;
    S_MFI_MNG_48 : S_MFI_MNG;
    S_MFI_MNG_49 : S_MFI_MNG;
    S_MFI_MNG_50 : S_MFI_MNG;
    S_MFI_MNG_51 : S_MFI_MNG;
    S_MFI_MNG_52 : S_MFI_MNG;
    S_MFI_MNG_53 : S_MFI_MNG;
    S_MFI_MNG_54 : S_MFI_MNG;
    S_MFI_MNG_55 : S_MFI_MNG;
    S_MFI_MNG_56 : S_MFI_MNG;
    S_MFI_MNG_57 : S_MFI_MNG;
    S_MFI_MNG_58 : S_MFI_MNG;
    S_MFI_MNG_59 : S_MFI_MNG;
    S_MFI_MNG_60 : S_MFI_MNG;
    S_MFI_MNG_61 : S_MFI_MNG;
    BatSyncUAct_Q : MFI;
    BatSocAct_Q : MFI;
    BmsHeartBeat_Q : MFI;
    BmsPartDiffVolt_Q : MFI;
    BatPNomMaxAct_Q : MFI;
    BmsDchrgMwhAct_Q : MFI;
    BmsCellMaxVolt_Q : MFI;
    BmsCellMinVolt_Q : MFI;
    BmsServSoC_Q : MFI;
    PSStateWord_Q : MFI;
    ABBStateWord_Q : MFI;
    GCPAct_Q : MFI;
    GCFAct_Q : MFI;
    GCSNomAct_Q : MFI;
    GCQAct_Q : MFI;
    GCPF_Q : MFI;
    GCEAct_Q : MFI;
    GCTempAct_Q : MFI;
    IGBTTempaAct_Q : MFI;
    TrafoTempAct_Q : MFI;
    OTTempAct_Q : MFI;
    GCUAct12_Q : MFI;
    GCUAct23_Q : MFI;
    GCUAct13_Q : MFI;
    GCUAct1N_Q : MFI;
    GCUAct2N_Q : MFI;
    GCUAct3N_Q : MFI;
    GCUAct_Q : MFI;
    GCABBErrorID_Q : MFI;
    GCSysFltCode_Q : MFI;
    BmsUdcAct_Q : MFI;
    BmsIdcAct_Q : MFI;
    BmsNomPAct_Q : MFI;
    BmsNomEAct_Q : MFI;
    BmsBatPNomMaxAct_Q : MFI;
    BmsBatPNomMinAct_Q : MFI;
    BmsPAct_Q : MFI;
    BmsEAct_Q : MFI;
    BmsSohAct_Q : MFI;
    BmsTempMaxAct_Q : MFI;
    BmsTempMinAct_Q : MFI;
    BmsSyncUSet_Q : MFI;
    BmsVersion_Q : MFI;
    BmsRacksNServiceCnt_Q : MFI;
    BmsTotalRackCnt_Q : MFI;
    BmsPartMinRackCnt_Q : MFI;
    S_MFI_MNG_62 : S_MFI_MNG;
    S_SPI_MNG_301 : S_SPI_MNG;
    S_SPI_MNG_302 : S_SPI_MNG;
    S_MFI_MNG_303 : S_MFI_MNG;
    S_MFI_MNG_304 : S_MFI_MNG;
    S_MFI_MNG_305 : S_MFI_MNG;
    S_MFI_MNG_306 : S_MFI_MNG;
    S_MFI_MNG_307 : S_MFI_MNG;
    S_SPI_MNG_308 : S_SPI_MNG;
    S_SPI_MNG_309 : S_SPI_MNG;
    S_MFI_MNG_310 : S_MFI_MNG;
    S_MFI_MNG_311 : S_MFI_MNG;
    S_MFI_MNG_312 : S_MFI_MNG;
    S_MFI_MNG_313 : S_MFI_MNG;
    S_MFI_MNG_314 : S_MFI_MNG;
    S_SPI_MNG_315 : S_SPI_MNG;
    S_SPI_MNG_316 : S_SPI_MNG;
    S_MFI_MNG_317 : S_MFI_MNG;
    S_MFI_MNG_318 : S_MFI_MNG;
    S_MFI_MNG_319 : S_MFI_MNG;
    S_MFI_MNG_320 : S_MFI_MNG;
    S_MFI_MNG_321 : S_MFI_MNG;
    S_SPI_MNG_322 : S_SPI_MNG;
    S_SPI_MNG_323 : S_SPI_MNG;
    S_MFI_MNG_324 : S_MFI_MNG;
    S_MFI_MNG_325 : S_MFI_MNG;
    S_MFI_MNG_326 : S_MFI_MNG;
    S_MFI_MNG_327 : S_MFI_MNG;
    S_MFI_MNG_328 : S_MFI_MNG;
    S_SPI_MNG_329 : S_SPI_MNG;
    S_SPI_MNG_330 : S_SPI_MNG;
    S_MFI_MNG_331 : S_MFI_MNG;
    S_MFI_MNG_332 : S_MFI_MNG;
    S_MFI_MNG_333 : S_MFI_MNG;
    S_MFI_MNG_334 : S_MFI_MNG;
    S_MFI_MNG_335 : S_MFI_MNG;
    S_SPI_MNG_336 : S_SPI_MNG;
    S_SPI_MNG_337 : S_SPI_MNG;
    S_MFI_MNG_338 : S_MFI_MNG;
    S_MFI_MNG_339 : S_MFI_MNG;
    S_MFI_MNG_340 : S_MFI_MNG;
    S_MFI_MNG_341 : S_MFI_MNG;
    S_MFI_MNG_342 : S_MFI_MNG;
    S_SPI_MNG_343 : S_SPI_MNG;
    S_SPI_MNG_344 : S_SPI_MNG;
    S_MFI_MNG_345 : S_MFI_MNG;
    S_MFI_MNG_346 : S_MFI_MNG;
    S_MFI_MNG_347 : S_MFI_MNG;
    S_MFI_MNG_348 : S_MFI_MNG;
    S_MFI_MNG_349 : S_MFI_MNG;
    S_SPI_MNG_350 : S_SPI_MNG;
    S_SPI_MNG_351 : S_SPI_MNG;
    S_MFI_MNG_352 : S_MFI_MNG;
    S_MFI_MNG_353 : S_MFI_MNG;
    S_MFI_MNG_354 : S_MFI_MNG;
    S_MFI_MNG_355 : S_MFI_MNG;
    S_MFI_MNG_356 : S_MFI_MNG;
    S_SPI_MNG_357 : S_SPI_MNG;
    S_SPI_MNG_358 : S_SPI_MNG;
    S_MFI_MNG_359 : S_MFI_MNG;
    S_MFI_MNG_360 : S_MFI_MNG;
    S_MFI_MNG_361 : S_MFI_MNG;
    S_MFI_MNG_362 : S_MFI_MNG;
    S_MFI_MNG_363 : S_MFI_MNG;
    S_SPI_MNG_364 : S_SPI_MNG;
    S_SPI_MNG_365 : S_SPI_MNG;
    S_MFI_MNG_366 : S_MFI_MNG;
    S_MFI_MNG_367 : S_MFI_MNG;
    S_MFI_MNG_368 : S_MFI_MNG;
    S_MFI_MNG_369 : S_MFI_MNG;
    S_MFI_MNG_370 : S_MFI_MNG;
    S_SPI_MNG_371 : S_SPI_MNG;
    S_SPI_MNG_372 : S_SPI_MNG;
    S_MFI_MNG_373 : S_MFI_MNG;
    S_MFI_MNG_374 : S_MFI_MNG;
    S_MFI_MNG_375 : S_MFI_MNG;
    S_MFI_MNG_376 : S_MFI_MNG;
    S_MFI_MNG_377 : S_MFI_MNG;
    S_SPI_MNG_378 : S_SPI_MNG;
    S_SPI_MNG_379 : S_SPI_MNG;
    S_MFI_MNG_380 : S_MFI_MNG;
    S_MFI_MNG_381 : S_MFI_MNG;
    S_MFI_MNG_382 : S_MFI_MNG;
    S_MFI_MNG_383 : S_MFI_MNG;
    S_MFI_MNG_384 : S_MFI_MNG;
    S_SPI_MNG_385 : S_SPI_MNG;
    S_SPI_MNG_386 : S_SPI_MNG;
    S_MFI_MNG_387 : S_MFI_MNG;
    S_MFI_MNG_388 : S_MFI_MNG;
    S_MFI_MNG_389 : S_MFI_MNG;
    S_MFI_MNG_390 : S_MFI_MNG;
    S_MFI_MNG_391 : S_MFI_MNG;
    S_SPI_MNG_392 : S_SPI_MNG;
    S_SPI_MNG_393 : S_SPI_MNG;
    S_MFI_MNG_394 : S_MFI_MNG;
    S_MFI_MNG_395 : S_MFI_MNG;
    S_MFI_MNG_396 : S_MFI_MNG;
    S_MFI_MNG_397 : S_MFI_MNG;
    S_MFI_MNG_398 : S_MFI_MNG;
    S_SPI_MNG_399 : S_SPI_MNG;
    S_SPI_MNG_400 : S_SPI_MNG;
    S_MFI_MNG_401 : S_MFI_MNG;
    S_MFI_MNG_402 : S_MFI_MNG;
    S_MFI_MNG_403 : S_MFI_MNG;
    S_MFI_MNG_404 : S_MFI_MNG;
    S_MFI_MNG_405 : S_MFI_MNG;
    S_SPI_MNG_406 : S_SPI_MNG;
    S_SPI_MNG_407 : S_SPI_MNG;
    S_MFI_MNG_408 : S_MFI_MNG;
    S_MFI_MNG_409 : S_MFI_MNG;
    S_MFI_MNG_410 : S_MFI_MNG;
    S_MFI_MNG_411 : S_MFI_MNG;
    S_MFI_MNG_412 : S_MFI_MNG;
    S_SPI_MNG_413 : S_SPI_MNG;
    S_SPI_MNG_414 : S_SPI_MNG;
    S_MFI_MNG_415 : S_MFI_MNG;
    S_MFI_MNG_416 : S_MFI_MNG;
    S_MFI_MNG_417 : S_MFI_MNG;
    S_MFI_MNG_418 : S_MFI_MNG;
    S_MFI_MNG_419 : S_MFI_MNG;
    S_SPI_MNG_420 : S_SPI_MNG;
    S_SPI_MNG_421 : S_SPI_MNG;
    S_MFI_MNG_422 : S_MFI_MNG;
    S_MFI_MNG_423 : S_MFI_MNG;
    S_MFI_MNG_424 : S_MFI_MNG;
    S_MFI_MNG_425 : S_MFI_MNG;
    S_MFI_MNG_426 : S_MFI_MNG;
    Rk1OnlineSt_Q : SPI;
    Rk1FaultSt_Q : SPI;
    Rk1SoCAct_Q : MFI;
    Rk1SoHAct_Q : MFI;
    Rk1UAct_Q : MFI;
    Rk1IAct_Q : MFI;
    Rk1TempAct_Q : MFI;
    Rk2OnlineSt_Q : SPI;
    Rk2FaultSt_Q : SPI;
    Rk2SoCAct_Q : MFI;
    Rk2SoHAct_Q : MFI;
    Rk2UAct_Q : MFI;
    Rk2IAct_Q : MFI;
    Rk2TempAct_Q : MFI;
    Rk3OnlineSt_Q : SPI;
    Rk3FaultSt_Q : SPI;
    Rk3SoCAct_Q : MFI;
    Rk3SoHAct_Q : MFI;
    Rk3UAct_Q : MFI;
    Rk3IAct_Q : MFI;
    Rk3TempAct_Q : MFI;
    Rk4OnlineSt_Q : SPI;
    Rk4FaultSt_Q : SPI;
    Rk4SoCAct_Q : MFI;
    Rk4SoHAct_Q : MFI;
    Rk4UAct_Q : MFI;
    Rk4IAct_Q : MFI;
    Rk4TempAct_Q : MFI;
    Rk5OnlineSt_Q : SPI;
    Rk5FaultSt_Q : SPI;
    Rk5SoCAct_Q : MFI;
    Rk5SoHAct_Q : MFI;
    Rk5UAct_Q : MFI;
    Rk5IAct_Q : MFI;
    Rk5TempAct_Q : MFI;
    Rk6OnlineSt_Q : SPI;
    Rk6FaultSt_Q : SPI;
    Rk6SoCAct_Q : MFI;
    Rk6SoHAct_Q : MFI;
    Rk6UAct_Q : MFI;
    Rk6IAct_Q : MFI;
    Rk6TempAct_Q : MFI;
    Rk7OnlineSt_Q : SPI;
    Rk7FaultSt_Q : SPI;
    Rk7SoCAct_Q : MFI;
    Rk7SoHAct_Q : MFI;
    Rk7UAct_Q : MFI;
    Rk7IAct_Q : MFI;
    Rk7TempAct_Q : MFI;
    Rk8OnlineSt_Q : SPI;
    Rk8FaultSt_Q : SPI;
    Rk8SoCAct_Q : MFI;
    Rk8SoHAct_Q : MFI;
    Rk8UAct_Q : MFI;
    Rk8IAct_Q : MFI;
    Rk8TempAct_Q : MFI;
    Rk9OnlineSt_Q : SPI;
    Rk9FaultSt_Q : SPI;
    Rk9SoCAct_Q : MFI;
    Rk9SoHAct_Q : MFI;
    Rk9UAct_Q : MFI;
    Rk9IAct_Q : MFI;
    Rk9TempAct_Q : MFI;
    Rk10OnlineSt_Q : SPI;
    Rk10FaultSt_Q : SPI;
    Rk10SoCAct_Q : MFI;
    Rk10SoHAct_Q : MFI;
    Rk10UAct_Q : MFI;
    Rk10IAct_Q : MFI;
    Rk10TempAct_Q : MFI;
    Rk11OnlineSt_Q : SPI;
    Rk11FaultSt_Q : SPI;
    Rk11SoCAct_Q : MFI;
    Rk11SoHAct_Q : MFI;
    Rk11UAct_Q : MFI;
    Rk11IAct_Q : MFI;
    Rk11TempAct_Q : MFI;
    Rk12OnlineSt_Q : SPI;
    Rk12FaultSt_Q : SPI;
    Rk12SoCAct_Q : MFI;
    Rk12SoHAct_Q : MFI;
    Rk12UAct_Q : MFI;
    Rk12IAct_Q : MFI;
    Rk12TempAct_Q : MFI;
    Rk13OnlineSt_Q : SPI;
    Rk13FaultSt_Q : SPI;
    Rk13SoCAct_Q : MFI;
    Rk13SoHAct_Q : MFI;
    Rk13UAct_Q : MFI;
    Rk13IAct_Q : MFI;
    Rk13TempAct_Q : MFI;
    Rk14OnlineSt_Q : SPI;
    Rk14FaultSt_Q : SPI;
    Rk14SoCAct_Q : MFI;
    Rk14SoHAct_Q : MFI;
    Rk14UAct_Q : MFI;
    Rk14IAct_Q : MFI;
    Rk14TempAct_Q : MFI;
    Rk15OnlineSt_Q : SPI;
    Rk15FaultSt_Q : SPI;
    Rk15SoCAct_Q : MFI;
    Rk15SoHAct_Q : MFI;
    Rk15UAct_Q : MFI;
    Rk15IAct_Q : MFI;
    Rk15TempAct_Q : MFI;
    Rk16OnlineSt_Q : SPI;
    Rk16FaultSt_Q : SPI;
    Rk16SoCAct_Q : MFI;
    Rk16SoHAct_Q : MFI;
    Rk16UAct_Q : MFI;
    Rk16IAct_Q : MFI;
    Rk16TempAct_Q : MFI;
    Rk17OnlineSt_Q : SPI;
    Rk17FaultSt_Q : SPI;
    Rk17SoCAct_Q : MFI;
    Rk17SoHAct_Q : MFI;
    Rk17UAct_Q : MFI;
    Rk17IAct_Q : MFI;
    Rk17TempAct_Q : MFI;
    Rk18OnlineSt_Q : SPI;
    Rk18FaultSt_Q : SPI;
    Rk18SoCAct_Q : MFI;
    Rk18SoHAct_Q : MFI;
    Rk18UAct_Q : MFI;
    Rk18IAct_Q : MFI;
    Rk18TempAct_Q : MFI;
    A252 : BOOL;
    A253 : BOOL;
    A254 : BOOL;
    A255 : BOOL;
    A256 : BOOL;
    A257 : BOOL;
    A258 : BOOL;
    A259 : BOOL;
    A260 : BOOL;
    A261 : BOOL;
    A262 : BOOL;
    A263 : BOOL;
    A264 : BOOL;
    A265 : BOOL;
    A266 : BOOL;
    A267 : BOOL;
    A268 : BOOL;
    A269 : BOOL;
    A270 : BOOL;
    A271 : BOOL;
    A272 : BOOL;
    A273 : BOOL;
    A274 : BOOL;
    A275 : BOOL;
    A276 : BOOL;
    A277 : BOOL;
    A278 : BOOL;
    A279 : BOOL;
    A280 : BOOL;
    A281 : BOOL;
    A282 : BOOL;
    A283 : BOOL;
    A284 : BOOL;
    A285 : BOOL;
    A286 : BOOL;
    A287 : BOOL;
    A288 : BOOL;
    A289 : BOOL;
    A290 : BOOL;
    A291 : BOOL;
    A292 : BOOL;
    A293 : BOOL;
    A294 : BOOL;
    A295 : BOOL;
    A296 : BOOL;
    A297 : BOOL;
    A298 : BOOL;
    A299 : BOOL;
    A300 : BOOL;
    A301 : BOOL;
    A302 : BOOL;
    A303 : BOOL;
    A304 : BOOL;
    A305 : BOOL;
    A306 : BOOL;
    A307 : BOOL;
    A308 : BOOL;
    A309 : BOOL;
    A310 : BOOL;
    A311 : BOOL;
    A312 : BOOL;
    A313 : BOOL;
    A314 : BOOL;
    A315 : BOOL;
    A316 : BOOL;
    A317 : BOOL;
    A318 : BOOL;
    A319 : BOOL;
    A320 : BOOL;
    A321 : BOOL;
    A322 : BOOL;
    A323 : BOOL;
    A324 : BOOL;
    A325 : BOOL;
    A326 : BOOL;
    A327 : BOOL;
    A328 : BOOL;
    A329 : BOOL;
    A330 : BOOL;
    A331 : BOOL;
    A332 : BOOL;
    A333 : BOOL;
    A334 : BOOL;
    A335 : BOOL;
    A336 : BOOL;
    A337 : BOOL;
    A338 : BOOL;
    A339 : BOOL;
    A340 : BOOL;
    A341 : BOOL;
    A342 : BOOL;
    A343 : BOOL;
    A344 : BOOL;
    A345 : BOOL;
    A346 : BOOL;
    A347 : BOOL;
    A348 : BOOL;
    A349 : BOOL;
    A350 : BOOL;
    A351 : BOOL;
    A352 : BOOL;
    A353 : BOOL;
    A354 : BOOL;
    A355 : BOOL;
    A356 : BOOL;
    A357 : BOOL;
    A358 : BOOL;
    A359 : BOOL;
    A360 : BOOL;
    A361 : BOOL;
    A362 : BOOL;
    A363 : BOOL;
    A364 : BOOL;
    A365 : BOOL;
    A366 : BOOL;
    A367 : BOOL;
    A368 : BOOL;
    A369 : BOOL;
    A370 : BOOL;
    A371 : BOOL;
    A372 : BOOL;
    A373 : BOOL;
    A374 : BOOL;
    A375 : BOOL;
    A376 : BOOL;
    A377 : BOOL;
    A378 : BOOL;
    A379 : BOOL;
    A380 : BOOL;
    A381 : BOOL;
    A382 : BOOL;
    A383 : BOOL;
    A384 : BOOL;
    A385 : BOOL;
    A386 : BOOL;
    A387 : BOOL;
    A388 : BOOL;
    A389 : BOOL;
    A390 : BOOL;
    A391 : BOOL;
    A392 : BOOL;
    A393 : BOOL;
    A394 : BOOL;
    A395 : BOOL;
    A396 : BOOL;
    A397 : BOOL;
    A398 : BOOL;
    A399 : BOOL;
    A400 : BOOL;
    A401 : BOOL;
    A402 : BOOL;
    A403 : BOOL;
    A404 : BOOL;
    A405 : BOOL;
    A406 : BOOL;
    A407 : BOOL;
    A408 : BOOL;
    A409 : BOOL;
    A410 : BOOL;
    A411 : BOOL;
    A412 : BOOL;
    A413 : BOOL;
    A414 : BOOL;
    A415 : BOOL;
    A416 : BOOL;
    A417 : BOOL;
    A418 : BOOL;
    A419 : BOOL;
    A420 : BOOL;
    A421 : BOOL;
    A422 : BOOL;
    A423 : BOOL;
    A424 : BOOL;
    A425 : BOOL;
    A426 : BOOL;
    A427 : BOOL;
    A428 : BOOL;
    A429 : BOOL;
    A430 : BOOL;
    A431 : BOOL;
    A432 : BOOL;
    A433 : BOOL;
    A434 : BOOL;
    A435 : BOOL;
    A436 : BOOL;
    A437 : BOOL;
    A438 : BOOL;
    A439 : BOOL;
    A440 : BOOL;
    A441 : BOOL;
    A442 : BOOL;
    A443 : BOOL;
    A444 : BOOL;
    A445 : BOOL;
    A446 : BOOL;
    A447 : BOOL;
    A448 : BOOL;
    A449 : BOOL;
    A450 : BOOL;
    A451 : BOOL;
    A452 : BOOL;
    A453 : BOOL;
    A454 : BOOL;
    A455 : BOOL;
    A456 : BOOL;
    A457 : BOOL;
    A458 : BOOL;
    A459 : BOOL;
    A460 : BOOL;
    A461 : BOOL;
    A462 : BOOL;
    A463 : BOOL;
    A464 : BOOL;
    A465 : BOOL;
    A466 : BOOL;
    A467 : BOOL;
    A468 : BOOL;
    A469 : BOOL;
    A470 : BOOL;
    A471 : BOOL;
    A472 : BOOL;
    A473 : BOOL;
    A474 : BOOL;
    A475 : BOOL;
    A476 : BOOL;
    A477 : BOOL;
    A478 : BOOL;
    A479 : BOOL;
    A480 : BOOL;
    A481 : BOOL;
    A482 : BOOL;
    A483 : BOOL;
    A484 : BOOL;
    A485 : BOOL;
    A486 : BOOL;
    A487 : BOOL;
    A488 : BOOL;
    A489 : BOOL;
    A490 : BOOL;
    A491 : BOOL;
    A492 : BOOL;
    A493 : BOOL;
    A494 : BOOL;
    A495 : BOOL;
    A496 : BOOL;
    A497 : BOOL;
    A498 : BOOL;
    A499 : BOOL;
    A500 : BOOL;
    emC_PPCOut_1 : emC_LuC_PPCOut;
    S_MFI_MNG_65 : S_MFI_MNG;
    GCIAvgAct_Q : MFI;
  END_VAR

						
							RTU_RTC_1(EN:=TRUE);
Timestamp.Milliseconds :=RTU_RTC_1.Milliseconds;
Timestamp.Minutes :=RTU_RTC_1.Minutes;
Timestamp.IV :=RTU_RTC_1.IV;
Timestamp.Hours :=RTU_RTC_1.Hours;
Timestamp.Summertime :=RTU_RTC_1.Summertime;
Timestamp.DayOfMonth :=RTU_RTC_1.DayOfMonth;
Timestamp.DayOfWeek :=RTU_RTC_1.DayOfWeek;
Timestamp.Month :=RTU_RTC_1.Months;
Timestamp.Year :=RTU_RTC_1.Year;
LUC_Num:=1;
							
							
								
								
